   1:  PR[91,2] = PR[90,2] + -1.776;
   1:L PR[91] R[100]mm/sec CNT100TB   .50sec,CALL END_PUD;
   1:  PR[92] = PR[91];
   1:  PR[92,3] = PR[92,3] + 20;
   1:J PR[92] 10% FINE;
   1:  PR[91] = PR[90];
   1:  PR[91,1] = PR[90,1] + 4.469;
   1:  PR[91,2] = PR[90,2] + -0.729;
   1:  PR[91,3] = PR[90,3] + 32.695;
   1:  PR[92] = PR[91];
   1:  PR[92,3] = PR[92,3] + 20;
   1:J PR[92] 10% FINE;
   1:L PR[91] R[100]mm/sec CNT100;
   1:  CALL LASER_DRAHT_START;
   1:  PR[91,1] = PR[90,1] + 5.143;
   1:  PR[91,2] = PR[90,2] + -5.829;
   1:L PR[91] R[100]mm/sec CNT100;
   1:  PR[91,1] = PR[90,1] + 7.118;
   1:  PR[91,2] = PR[90,2] + -10.577;
   1:L PR[91] R[100]mm/sec CNT100;
   1:  PR[91,1] = PR[90,1] + 10.256;
   1:  PR[91,2] = PR[90,2] + -14.648;
   1:L PR[91] R[100]mm/sec CNT100;
   1:  PR[91,1] = PR[90,1] + 14.340;
   1:  PR[91,2] = PR[90,2] + -17.763;
   1:L PR[91] R[100]mm/sec CNT100;
   1:  PR[91,1] = PR[90,1] + 17.726;
   1:  PR[91,2] = PR[90,2] + -19.159;
   1:L PR[91] R[100]mm/sec CNT100;
   1:  PR[91,1] = PR[90,1] + 19.081;
   1:  PR[91,2] = PR[90,2] + -19.714;
   1:L PR[91] R[100]mm/sec CNT100;
   1:  PR[91,1] = PR[90,1] + 24.162;
   1:  PR[91,2] = PR[90,2] + -20.375;
   1:L PR[91] R[100]mm/sec CNT100;
   1:  PR[91,1] = PR[90,1] + 29.234;
   1:  PR[91,2] = PR[90,2] + -19.704;
   1:L PR[91] R[100]mm/sec CNT100;
   1:  PR[91,1] = PR[90,1] + 32.324;
   1:  PR[91,2] = PR[90,2] + -18.438;
   1:L PR[91] R[100]mm/sec CNT100;
   1:  PR[91,1] = PR[90,1] + 33.950;
   1:  PR[91,2] = PR[90,2] + -17.758;
   1:L PR[91] R[100]mm/sec CNT100;
   1:  PR[91,1] = PR[90,1] + 36.544;
   1:  PR[91,2] = PR[90,2] + -15.795;
   1:L PR[91] R[100]mm/sec CNT100;
   1:  PR[91,1] = PR[90,1] + 38.003;
   1:  PR[91,2] = PR[90,2] + -14.670;
   1:L PR[91] R[100]mm/sec CNT100;
   1:  PR[91,1] = PR[90,1] + 39.978;
   1:  PR[91,2] = PR[90,2] + -12.142;
   1:L PR[91] R[100]mm/sec CNT100;
   1:  PR[91,1] = PR[90,1] + 41.183;
   1:  PR[91,2] = PR[90,2] + -10.565;
   1:L PR[91] R[100]mm/sec CNT100;
   1:  PR[91,1] = PR[90,1] + 41.364;
   1:  PR[91,2] = PR[90,2] + -10.235;
   1:L PR[91] R[100]mm/sec CNT100;
   1:  PR[91,1] = PR[90,1] + 42.070;
   1:  PR[91,2] = PR[90,2] + -8.524;
   1:L PR[91] R[100]mm/sec CNT100;
   1:  PR[91,1] = PR[90,1] + 42.766;
   1:  PR[91,2] = PR[90,2] + -6.971;
   1:L PR[91] R[100]mm/sec CNT100;
   1:  PR[91,1] = PR[90,1] + 43.473;
   1:  PR[91,2] = PR[90,2] + -4.203;
   1:L PR[91] R[100]mm/sec CNT100;
   1:  PR[91,1] = PR[90,1] + 43.657;
   1:  PR[91,2] = PR[90,2] + -2.266;
   1:L PR[91] R[100]mm/sec CNT100;
   1:  PR[91,1] = PR[90,1] + 47.140;
   1:  PR[91,2] = PR[90,2] + -2.119;
   1:L PR[91] R[100]mm/sec CNT100;
   1:  PR[91,1] = PR[90,1] + 47.551;
   1:  PR[91,2] = PR[90,2] + -4.387;
   1:L PR[91] R[100]mm/sec CNT100;
   1:  PR[91,1] = PR[90,1] + 47.975;
   1:  PR[91,2] = PR[90,2] + -5.947;
   1:L PR[91] R[100]mm/sec CNT100;
   1:  PR[91,1] = PR[90,1] + 48.962;
   1:  PR[91,2] = PR[90,2] + -7.849;
   1:L PR[91] R[100]mm/sec CNT100;
   1:  PR[91,1] = PR[90,1] + 50.226;
   1:  PR[91,2] = PR[90,2] + -10.536;
   1:L PR[91] R[100]mm/sec CNT100;
   1:  PR[91,1] = PR[90,1] + 50.408;
   1:  PR[91,2] = PR[90,2] + -10.773;
   1:L PR[91] R[100]mm/sec CNT100;
   1:  PR[91,1] = PR[90,1] + 53.451;
   1:  PR[91,2] = PR[90,2] + -14.307;
   1:L PR[91] R[100]mm/sec CNT100;
   1:  PR[91,1] = PR[90,1] + 54.867;
   1:  PR[91,2] = PR[90,2] + -15.442;
   1:L PR[91] R[100]mm/sec CNT100;
   1:  PR[91,1] = PR[90,1] + 57.318;
   1:  PR[91,2] = PR[90,2] + -17.146;
   1:L PR[91] R[100]mm/sec CNT100;
   1:  PR[91,1] = PR[90,1] + 60.422;
   1:  PR[91,2] = PR[90,2] + -18.651;
   1:L PR[91] R[100]mm/sec CNT100;
   1:  PR[91,1] = PR[90,1] + 61.529;
   1:  PR[91,2] = PR[90,2] + -19.083;
   1:L PR[91] R[100]mm/sec CNT100;
   1:  PR[91,1] = PR[90,1] + 65.504;
   1:  PR[91,2] = PR[90,2] + -20.053;
   1:L PR[91] R[100]mm/sec CNT100;
   1:  PR[91,1] = PR[90,1] + 66.069;
   1:  PR[91,2] = PR[90,2] + -20.209;
   1:L PR[91] R[100]mm/sec CNT100;
   1:  PR[91,1] = PR[90,1] + 70.771;
   1:  PR[91,2] = PR[90,2] + -20.477;
   1:L PR[91] R[100]mm/sec CNT100;
   1:  PR[91,1] = PR[90,1] + 71.856;
   1:  PR[91,2] = PR[90,2] + -20.322;
   1:L PR[91] R[100]mm/sec CNT100;
   1:  PR[91,1] = PR[90,1] + 75.350;
   1:  PR[91,2] = PR[90,2] + -19.774;
   1:L PR[91] R[100]mm/sec CNT100;
   1:  PR[91,1] = PR[90,1] + 77.247;
   1:  PR[91,2] = PR[90,2] + -19.075;
   1:L PR[91] R[100]mm/sec CNT100;
   1:  PR[91,1] = PR[90,1] + 79.618;
   1:  PR[91,2] = PR[90,2] + -18.166;
   1:L PR[91] R[100]mm/sec CNT100;
   1:  PR[91,1] = PR[90,1] + 81.915;
   1:  PR[91,2] = PR[90,2] + -16.702;
   1:L PR[91] R[100]mm/sec CNT100;
   1:  PR[91,1] = PR[90,1] + 83.382;
   1:  PR[91,2] = PR[90,2] + -15.743;
   1:L PR[91] R[100]mm/sec CNT100;
   1:  PR[91,1] = PR[90,1] + 86.493;
   1:  PR[91,2] = PR[90,2] + -12.622;
   1:L PR[91] R[100]mm/sec CNT100;
   1:  PR[91,1] = PR[90,1] + 88.806;
   1:  PR[91,2] = PR[90,2] + -8.967;
   1:L PR[91] R[100]mm/sec CNT100;
   1:  PR[91,1] = PR[90,1] + 90.231;
   1:  PR[91,2] = PR[90,2] + -4.940;
   1:L PR[91] R[100]mm/sec CNT100;
   1:  PR[91,1] = PR[90,1] + 90.718;
   1:  PR[91,2] = PR[90,2] + -0.729;
   1:L PR[91] R[100]mm/sec CNT100;
   1:  PR[91,1] = PR[90,1] + 90.231;
   1:  PR[91,2] = PR[90,2] + 3.481;
   1:L PR[91] R[100]mm/sec CNT100;
   1:  PR[91,1] = PR[90,1] + 88.806;
   1:  PR[91,2] = PR[90,2] + 7.508;
   1:L PR[91] R[100]mm/sec CNT100;
   1:  PR[91,1] = PR[90,1] + 86.495;
   1:  PR[91,2] = PR[90,2] + 11.160;
   1:L PR[91] R[100]mm/sec CNT100;
   1:  PR[91,1] = PR[90,1] + 84.284;
   1:  PR[91,2] = PR[90,2] + 13.362;
   1:L PR[91] R[100]mm/sec CNT100;
   1:  PR[91,1] = PR[90,1] + 83.384;
   1:  PR[91,2] = PR[90,2] + 14.279;
   1:L PR[91] R[100]mm/sec CNT100;
   1:  PR[91,1] = PR[90,1] + 81.098;
   1:  PR[91,2] = PR[90,2] + 15.732;
   1:L PR[91] R[100]mm/sec CNT100;
   1:  PR[91,1] = PR[90,1] + 79.618;
   1:  PR[91,2] = PR[90,2] + 16.704;
   1:L PR[91] R[100]mm/sec CNT100;
   1:  PR[91,1] = PR[90,1] + 77.562;
   1:  PR[91,2] = PR[90,2] + 17.457;
   1:L PR[91] R[100]mm/sec CNT100;
   1:  PR[91,1] = PR[90,1] + 75.350;
   1:  PR[91,2] = PR[90,2] + 18.312;
   1:L PR[91] R[100]mm/sec CNT100;
   1:  PR[91,1] = PR[90,1] + 73.814;
   1:  PR[91,2] = PR[90,2] + 18.527;
   1:L PR[91] R[100]mm/sec CNT100;
   1:  PR[91,1] = PR[90,1] + 70.770;
   1:  PR[91,2] = PR[90,2] + 19.014;
   1:L PR[91] R[100]mm/sec CNT100;
   1:  PR[91,1] = PR[90,1] + 69.982;
   1:  PR[91,2] = PR[90,2] + 18.956;
   1:L PR[91] R[100]mm/sec CNT100;
   1:  PR[91,1] = PR[90,1] + 66.065;
   1:  PR[91,2] = PR[90,2] + 18.749;
   1:L PR[91] R[100]mm/sec CNT100;
   1:  PR[91,1] = PR[90,1] + 65.504;
   1:  PR[91,2] = PR[90,2] + 18.594;
   1:L PR[91] R[100]mm/sec CNT100;
   1:  PR[91,1] = PR[90,1] + 61.529;
   1:  PR[91,2] = PR[90,2] + 17.625;
   1:L PR[91] R[100]mm/sec CNT100;
   1:  PR[91,1] = PR[90,1] + 60.422;
   1:  PR[91,2] = PR[90,2] + 17.192;
   1:L PR[91] R[100]mm/sec CNT100;
   1:  PR[91,1] = PR[90,1] + 57.318;
   1:  PR[91,2] = PR[90,2] + 15.687;
   1:L PR[91] R[100]mm/sec CNT100;
   1:  PR[91,1] = PR[90,1] + 54.868;
   1:  PR[91,2] = PR[90,2] + 13.984;
   1:L PR[91] R[100]mm/sec CNT100;
   1:  PR[91,1] = PR[90,1] + 53.452;
   1:  PR[91,2] = PR[90,2] + 12.849;
   1:L PR[91] R[100]mm/sec CNT100;
   1:  PR[91,1] = PR[90,1] + 50.409;
   1:  PR[91,2] = PR[90,2] + 9.316;
   1:L PR[91] R[100]mm/sec CNT100;
   1:  PR[91,1] = PR[90,1] + 50.226;
   1:  PR[91,2] = PR[90,2] + 9.078;
   1:L PR[91] R[100]mm/sec CNT100;
   1:  PR[91,1] = PR[90,1] + 48.961;
   1:  PR[91,2] = PR[90,2] + 6.389;
   1:L PR[91] R[100]mm/sec CNT100;
   1:  PR[91,1] = PR[90,1] + 47.985;
   1:  PR[91,2] = PR[90,2] + 4.511;
   1:L PR[91] R[100]mm/sec CNT100;
   1:  PR[91,1] = PR[90,1] + 47.482;
   1:  PR[91,2] = PR[90,2] + 2.646;
   1:L PR[91] R[100]mm/sec CNT100;
   1:  PR[91,1] = PR[90,1] + 47.137;
   1:  PR[91,2] = PR[90,2] + 0.760;
   1:L PR[91] R[100]mm/sec CNT100;
   1:  PR[91,1] = PR[90,1] + 43.653;
   1:  PR[91,2] = PR[90,2] + 0.914;
   1:L PR[91] R[100]mm/sec CNT100;
   1:  PR[91,1] = PR[90,1] + 43.495;
   1:  PR[91,2] = PR[90,2] + 2.623;
   1:L PR[91] R[100]mm/sec CNT100;
   1:  PR[91,1] = PR[90,1] + 42.693;
   1:  PR[91,2] = PR[90,2] + 5.724;
   1:L PR[91] R[100]mm/sec CNT100;
   1:  PR[91,1] = PR[90,1] + 42.326;
   1:  PR[91,2] = PR[90,2] + 6.613;
   1:L PR[91] R[100]mm/sec CNT100;
   1:  PR[91,1] = PR[90,1] + 41.404;
   1:  PR[91,2] = PR[90,2] + 8.700;
   1:L PR[91] R[100]mm/sec CNT100;
   1:  PR[91,1] = PR[90,1] + 41.184;
   1:  PR[91,2] = PR[90,2] + 9.104;
   1:L PR[91] R[100]mm/sec CNT100;
   1:  PR[91,1] = PR[90,1] + 39.948;
   1:  PR[91,2] = PR[90,2] + 10.732;
   1:L PR[91] R[100]mm/sec CNT100;
   1:  PR[91,1] = PR[90,1] + 37.982;
   1:  PR[91,2] = PR[90,2] + 13.232;
   1:L PR[91] R[100]mm/sec CNT100;
   1:  PR[91,1] = PR[90,1] + 36.524;
   1:  PR[91,2] = PR[90,2] + 14.357;
   1:L PR[91] R[100]mm/sec CNT100;
   1:  PR[91,1] = PR[90,1] + 33.926;
   1:  PR[91,2] = PR[90,2] + 16.313;
   1:L PR[91] R[100]mm/sec CNT100;
   1:  PR[91,1] = PR[90,1] + 32.300;
   1:  PR[91,2] = PR[90,2] + 16.993;
   1:L PR[91] R[100]mm/sec CNT100;
   1:  PR[91,1] = PR[90,1] + 29.208;
   1:  PR[91,2] = PR[90,2] + 18.253;
   1:L PR[91] R[100]mm/sec CNT100;
   1:  PR[91,1] = PR[90,1] + 27.552;
   1:  PR[91,2] = PR[90,2] + 18.478;
   1:L PR[91] R[100]mm/sec CNT100;
   1:  PR[91,1] = PR[90,1] + 24.143;
   1:  PR[91,2] = PR[90,2] + 18.917;
   1:L PR[91] R[100]mm/sec CNT100;
   1:  PR[91,1] = PR[90,1] + 19.065;
   1:  PR[91,2] = PR[90,2] + 18.251;
   1:L PR[91] R[100]mm/sec CNT100;
   1:  PR[91,1] = PR[90,1] + 14.324;
   1:  PR[91,2] = PR[90,2] + 16.295;
   1:L PR[91] R[100]mm/sec CNT100;
   1:  PR[91,1] = PR[90,1] + 13.237;
   1:  PR[91,2] = PR[90,2] + 15.467;
   1:L PR[91] R[100]mm/sec CNT100;
   1:  PR[91,1] = PR[90,1] + 10.248;
   1:  PR[91,2] = PR[90,2] + 13.181;
   1:L PR[91] R[100]mm/sec CNT100;
   1:  PR[91,1] = PR[90,1] + 7.114;
   1:  PR[91,2] = PR[90,2] + 9.111;
   1:L PR[91] R[100]mm/sec CNT100;
   1:  PR[91,1] = PR[90,1] + 5.142;
   1:  PR[91,2] = PR[90,2] + 4.367;
   1:L PR[91] R[100]mm/sec CNT100;
   1:  PR[91,1] = PR[90,1] + 4.469;
   1:  PR[91,2] = PR[90,2] + -0.729;
   1:L PR[91] R[100]mm/sec CNT100TB   .50sec,CALL END_PUD;
   1:  PR[92] = PR[91];
   1:  PR[92,3] = PR[92,3] + 20;
   1:J PR[92] 10% FINE;
   1:  PR[91,1] = PR[90,1] + -41.681;
   1:  PR[91,2] = PR[90,2] + -0.717;
   1:  PR[92] = PR[91];
   1:  PR[92,3] = PR[92,3] + 20;
   1:J PR[92] 10% FINE;
   1:L PR[91] R[100]mm/sec CNT100;
   1:  CALL LASER_DRAHT_START;
   1:  PR[91,1] = PR[90,1] + -41.546;
   1:  PR[91,2] = PR[90,2] + -1.807;
   1:L PR[91] R[100]mm/sec CNT100;
   1:  PR[91,1] = PR[90,1] + -41.199;
   1:  PR[91,2] = PR[90,2] + -4.905;
   1:L PR[91] R[100]mm/sec CNT100;
   1:  PR[91,1] = PR[90,1] + -39.815;
   1:  PR[91,2] = PR[90,2] + -8.880;
   1:L PR[91] R[100]mm/sec CNT100;
   1:  PR[91,1] = PR[90,1] + -37.577;
   1:  PR[91,2] = PR[90,2] + -12.464;
   1:L PR[91] R[100]mm/sec CNT100;
   1:  PR[91,1] = PR[90,1] + -34.591;
   1:  PR[91,2] = PR[90,2] + -15.481;
   1:L PR[91] R[100]mm/sec CNT100;
   1:  PR[91,1] = PR[90,1] + -30.997;
   1:  PR[91,2] = PR[90,2] + -17.783;
   1:L PR[91] R[100]mm/sec CNT100;
   1:  PR[91,1] = PR[90,1] + -26.963;
   1:  PR[91,2] = PR[90,2] + -19.248;
   1:L PR[91] R[100]mm/sec CNT100;
   1:  PR[91,1] = PR[90,1] + -22.671;
   1:  PR[91,2] = PR[90,2] + -19.803;
   1:L PR[91] R[100]mm/sec CNT100;
   1:  PR[91,1] = PR[90,1] + -18.279;
   1:  PR[91,2] = PR[90,2] + -19.439;
   1:L PR[91] R[100]mm/sec CNT100;
   1:  PR[91,1] = PR[90,1] + -18.066;
   1:  PR[91,2] = PR[90,2] + -19.387;
   1:L PR[91] R[100]mm/sec CNT100;
   1:  PR[91,1] = PR[90,1] + -14.122;
   1:  PR[91,2] = PR[90,2] + -18.164;
   1:L PR[91] R[100]mm/sec CNT100;
   1:  PR[91,1] = PR[90,1] + -13.522;
   1:  PR[91,2] = PR[90,2] + -17.867;
   1:L PR[91] R[100]mm/sec CNT100;
   1:  PR[91,1] = PR[90,1] + -10.339;
   1:  PR[91,2] = PR[90,2] + -16.033;
   1:L PR[91] R[100]mm/sec CNT100;
   1:  PR[91,1] = PR[90,1] + -9.487;
   1:  PR[91,2] = PR[90,2] + -15.341;
   1:L PR[91] R[100]mm/sec CNT100;
   1:  PR[91,1] = PR[90,1] + -7.115;
   1:  PR[91,2] = PR[90,2] + -13.139;
   1:L PR[91] R[100]mm/sec CNT100;
   1:  PR[91,1] = PR[90,1] + -6.219;
   1:  PR[91,2] = PR[90,2] + -11.981;
   1:L PR[91] R[100]mm/sec CNT100;
   1:  PR[91,1] = PR[90,1] + -4.619;
   1:  PR[91,2] = PR[90,2] + -9.603;
   1:L PR[91] R[100]mm/sec CNT100;
   1:  PR[91,1] = PR[90,1] + -3.902;
   1:  PR[91,2] = PR[90,2] + -8.021;
   1:L PR[91] R[100]mm/sec CNT100;
   1:  PR[91,1] = PR[90,1] + -2.996;
   1:  PR[91,2] = PR[90,2] + -5.591;
   1:L PR[91] R[100]mm/sec CNT100;
   1:  PR[91,1] = PR[90,1] + -2.643;
   1:  PR[91,2] = PR[90,2] + -3.715;
   1:L PR[91] R[100]mm/sec CNT100;
   1:  PR[91,1] = PR[90,1] + -2.344;
   1:  PR[91,2] = PR[90,2] + -1.237;
   1:L PR[91] R[100]mm/sec CNT100;
   1:  PR[91,1] = PR[90,1] + -2.332;
   1:  PR[91,2] = PR[90,2] + -0.821;
   1:L PR[91] R[100]mm/sec CNT100;
   1:  PR[91,1] = PR[90,1] + -2.639;
   1:  PR[91,2] = PR[90,2] + 1.729;
   1:L PR[91] R[100]mm/sec CNT100;
   1:  PR[91,1] = PR[90,1] + -2.659;
   1:  PR[91,2] = PR[90,2] + 2.337;
   1:L PR[91] R[100]mm/sec CNT100;
   1:  PR[91,1] = PR[90,1] + -2.994;
   1:  PR[91,2] = PR[90,2] + 4.125;
   1:L PR[91] R[100]mm/sec CNT100;
   1:  PR[91,1] = PR[90,1] + -3.900;
   1:  PR[91,2] = PR[90,2] + 6.556;
   1:L PR[91] R[100]mm/sec CNT100;
   1:  PR[91,1] = PR[90,1] + -4.616;
   1:  PR[91,2] = PR[90,2] + 8.139;
   1:L PR[91] R[100]mm/sec CNT100;
   1:  PR[91,1] = PR[90,1] + -6.216;
   1:  PR[91,2] = PR[90,2] + 10.518;
   1:L PR[91] R[100]mm/sec CNT100;
   1:  PR[91,1] = PR[90,1] + -7.112;
   1:  PR[91,2] = PR[90,2] + 11.677;
   1:L PR[91] R[100]mm/sec CNT100;
   1:  PR[91,1] = PR[90,1] + -9.484;
   1:  PR[91,2] = PR[90,2] + 13.879;
   1:L PR[91] R[100]mm/sec CNT100;
   1:  PR[91,1] = PR[90,1] + -10.336;
   1:  PR[91,2] = PR[90,2] + 14.573;
   1:L PR[91] R[100]mm/sec CNT100;
   1:  PR[91,1] = PR[90,1] + -13.520;
   1:  PR[91,2] = PR[90,2] + 16.407;
   1:L PR[91] R[100]mm/sec CNT100;
   1:  PR[91,1] = PR[90,1] + -14.120;
   1:  PR[91,2] = PR[90,2] + 16.705;
   1:L PR[91] R[100]mm/sec CNT100;
   1:  PR[91,1] = PR[90,1] + -18.065;
   1:  PR[91,2] = PR[90,2] + 17.927;
   1:L PR[91] R[100]mm/sec CNT100;
   1:  PR[91,1] = PR[90,1] + -18.278;
   1:  PR[91,2] = PR[90,2] + 17.980;
   1:L PR[91] R[100]mm/sec CNT100;
   1:  PR[91,1] = PR[90,1] + -22.679;
   1:  PR[91,2] = PR[90,2] + 18.344;
   1:L PR[91] R[100]mm/sec CNT100;
   1:  PR[91,1] = PR[90,1] + -26.963;
   1:  PR[91,2] = PR[90,2] + 17.790;
   1:L PR[91] R[100]mm/sec CNT100;
   1:  PR[91,1] = PR[90,1] + -30.997;
   1:  PR[91,2] = PR[90,2] + 16.324;
   1:L PR[91] R[100]mm/sec CNT100;
   1:  PR[91,1] = PR[90,1] + -34.591;
   1:  PR[91,2] = PR[90,2] + 14.022;
   1:L PR[91] R[100]mm/sec CNT100;
   1:  PR[91,1] = PR[90,1] + -37.577;
   1:  PR[91,2] = PR[90,2] + 11.005;
   1:L PR[91] R[100]mm/sec CNT100;
   1:  PR[91,1] = PR[90,1] + -39.815;
   1:  PR[91,2] = PR[90,2] + 7.422;
   1:L PR[91] R[100]mm/sec CNT100;
   1:  PR[91,1] = PR[90,1] + -41.199;
   1:  PR[91,2] = PR[90,2] + 3.445;
   1:L PR[91] R[100]mm/sec CNT100;
   1:  PR[91,1] = PR[90,1] + -41.330;
   1:  PR[91,2] = PR[90,2] + 2.291;
   1:L PR[91] R[100]mm/sec CNT100;
   1:  PR[91,1] = PR[90,1] + -41.361;
   1:  PR[91,2] = PR[90,2] + 2.140;
   1:L PR[91] R[100]mm/sec CNT100;
   1:  PR[91,1] = PR[90,1] + -41.681;
   1:  PR[91,2] = PR[90,2] + -0.717;
   1:L PR[91] R[100]mm/sec CNT100TB   .50sec,CALL END_PUD;
   1:  PR[92] = PR[91];
   1:  PR[92,3] = PR[92,3] + 20;
   1:J PR[92] 10% FINE;
   1:  PR[91,1] = PR[90,1] + -77.314;
   1:  PR[91,2] = PR[90,2] + -18.642;
   1:  PR[92] = PR[91];
   1:  PR[92,3] = PR[92,3] + 20;
   1:J PR[92] 10% FINE;
   1:L PR[91] R[100]mm/sec CNT100;
   1:  CALL LASER_DRAHT_START;
   1:  PR[91,1] = PR[90,1] + -74.683;
   1:  PR[91,2] = PR[90,2] + -19.231;
   1:L PR[91] R[100]mm/sec CNT100;
   1:  PR[91,1] = PR[90,1] + -73.251;
   1:  PR[91,2] = PR[90,2] + -19.573;
   1:L PR[91] R[100]mm/sec CNT100;
   1:  PR[91,1] = PR[90,1] + -71.069;
   1:  PR[91,2] = PR[90,2] + -19.621;
   1:L PR[91] R[100]mm/sec CNT100;
   1:  PR[91,1] = PR[90,1] + -69.047;
   1:  PR[91,2] = PR[90,2] + -19.694;
   1:L PR[91] R[100]mm/sec CNT100;
   1:  PR[91,1] = PR[90,1] + -67.474;
   1:  PR[91,2] = PR[90,2] + -19.413;
   1:L PR[91] R[100]mm/sec CNT100;
   1:  PR[91,1] = PR[90,1] + -64.878;
   1:  PR[91,2] = PR[90,2] + -18.989;
   1:L PR[91] R[100]mm/sec CNT100;
   1:  PR[91,1] = PR[90,1] + -63.990;
   1:  PR[91,2] = PR[90,2] + -18.636;
   1:L PR[91] R[100]mm/sec CNT100;
   1:  PR[91,1] = PR[90,1] + -60.914;
   1:  PR[91,2] = PR[90,2] + -17.467;
   1:L PR[91] R[100]mm/sec CNT100;
   1:  PR[91,1] = PR[90,1] + -58.205;
   1:  PR[91,2] = PR[90,2] + -15.726;
   1:L PR[91] R[100]mm/sec CNT100;
   1:  PR[91,1] = PR[90,1] + -57.250;
   1:  PR[91,2] = PR[90,2] + -15.156;
   1:L PR[91] R[100]mm/sec CNT100;
   1:  PR[91,1] = PR[90,1] + -54.565;
   1:  PR[91,2] = PR[90,2] + -12.649;
   1:L PR[91] R[100]mm/sec CNT100;
   1:  PR[91,1] = PR[90,1] + -54.071;
   1:  PR[91,2] = PR[90,2] + -12.203;
   1:L PR[91] R[100]mm/sec CNT100;
   1:  PR[91,1] = PR[90,1] + -52.386;
   1:  PR[91,2] = PR[90,2] + -9.733;
   1:L PR[91] R[100]mm/sec CNT100;
   1:  PR[91,1] = PR[90,1] + -51.665;
   1:  PR[91,2] = PR[90,2] + -8.704;
   1:L PR[91] R[100]mm/sec CNT100;
   1:  PR[91,1] = PR[90,1] + -50.168;
   1:  PR[91,2] = PR[90,2] + -4.823;
   1:L PR[91] R[100]mm/sec CNT100;
   1:  PR[91,1] = PR[90,1] + -49.910;
   1:  PR[91,2] = PR[90,2] + -2.744;
   1:L PR[91] R[100]mm/sec CNT100;
   1:  PR[91,1] = PR[90,1] + -49.770;
   1:  PR[91,2] = PR[90,2] + -0.743;
   1:L PR[91] R[100]mm/sec CNT100;
   1:  PR[91,1] = PR[90,1] + -49.798;
   1:  PR[91,2] = PR[90,2] + -0.406;
   1:L PR[91] R[100]mm/sec CNT100;
   1:  PR[91,1] = PR[90,1] + -50.252;
   1:  PR[91,2] = PR[90,2] + 3.373;
   1:L PR[91] R[100]mm/sec CNT100;
   1:  PR[91,1] = PR[90,1] + -51.720;
   1:  PR[91,2] = PR[90,2] + 7.273;
   1:L PR[91] R[100]mm/sec CNT100;
   1:  PR[91,1] = PR[90,1] + -52.373;
   1:  PR[91,2] = PR[90,2] + 8.257;
   1:L PR[91] R[100]mm/sec CNT100;
   1:  PR[91,1] = PR[90,1] + -54.073;
   1:  PR[91,2] = PR[90,2] + 10.775;
   1:L PR[91] R[100]mm/sec CNT100;
   1:  PR[91,1] = PR[90,1] + -55.593;
   1:  PR[91,2] = PR[90,2] + 12.234;
   1:L PR[91] R[100]mm/sec CNT100;
   1:  PR[91,1] = PR[90,1] + -57.173;
   1:  PR[91,2] = PR[90,2] + 13.722;
   1:L PR[91] R[100]mm/sec CNT100;
   1:  PR[91,1] = PR[90,1] + -60.872;
   1:  PR[91,2] = PR[90,2] + 15.996;
   1:L PR[91] R[100]mm/sec CNT100;
   1:  PR[91,1] = PR[90,1] + -64.984;
   1:  PR[91,2] = PR[90,2] + 17.505;
   1:L PR[91] R[100]mm/sec CNT100;
   1:  PR[91,1] = PR[90,1] + -69.137;
   1:  PR[91,2] = PR[90,2] + 18.221;
   1:L PR[91] R[100]mm/sec CNT100;
   1:  PR[91,1] = PR[90,1] + -73.297;
   1:  PR[91,2] = PR[90,2] + 18.107;
   1:L PR[91] R[100]mm/sec CNT100;
   1:  PR[91,1] = PR[90,1] + -77.320;
   1:  PR[91,2] = PR[90,2] + 17.184;
   1:L PR[91] R[100]mm/sec CNT100;
   1:  PR[91,1] = PR[90,1] + -81.037;
   1:  PR[91,2] = PR[90,2] + 15.500;
   1:L PR[91] R[100]mm/sec CNT100;
   1:  PR[91,1] = PR[90,1] + -84.300;
   1:  PR[91,2] = PR[90,2] + 13.138;
   1:L PR[91] R[100]mm/sec CNT100;
   1:  PR[91,1] = PR[90,1] + -86.977;
   1:  PR[91,2] = PR[90,2] + 10.199;
   1:L PR[91] R[100]mm/sec CNT100;
   1:  PR[91,1] = PR[90,1] + -88.967;
   1:  PR[91,2] = PR[90,2] + 6.813;
   1:L PR[91] R[100]mm/sec CNT100;
   1:  PR[91,1] = PR[90,1] + -90.190;
   1:  PR[91,2] = PR[90,2] + 3.119;
   1:L PR[91] R[100]mm/sec CNT100;
   1:  PR[91,1] = PR[90,1] + -90.556;
   1:  PR[91,2] = PR[90,2] + -0.259;
   1:L PR[91] R[100]mm/sec CNT100;
   1:  PR[91,1] = PR[90,1] + -90.654;
   1:  PR[91,2] = PR[90,2] + -0.746;
   1:L PR[91] R[100]mm/sec CNT100;
   1:  PR[91,1] = PR[90,1] + -90.252;
   1:  PR[91,2] = PR[90,2] + -4.584;
   1:L PR[91] R[100]mm/sec CNT100;
   1:  PR[91,1] = PR[90,1] + -89.055;
   1:  PR[91,2] = PR[90,2] + -8.268;
   1:L PR[91] R[100]mm/sec CNT100;
   1:  PR[91,1] = PR[90,1] + -87.060;
   1:  PR[91,2] = PR[90,2] + -11.645;
   1:L PR[91] R[100]mm/sec CNT100;
   1:  PR[91,1] = PR[90,1] + -84.363;
   1:  PR[91,2] = PR[90,2] + -14.584;
   1:L PR[91] R[100]mm/sec CNT100;
   1:  PR[91,1] = PR[90,1] + -81.074;
   1:  PR[91,2] = PR[90,2] + -16.950;
   1:L PR[91] R[100]mm/sec CNT100;
   1:  PR[91,1] = PR[90,1] + -78.209;
   1:  PR[91,2] = PR[90,2] + -18.229;
   1:L PR[91] R[100]mm/sec CNT100;
   1:  PR[91,1] = PR[90,1] + -77.314;
   1:  PR[91,2] = PR[90,2] + -18.642;
   1:L PR[91] R[100]mm/sec CNT100TB   .50sec,CALL END_PUD;
   1:  PR[92] = PR[91];
   1:  PR[92,3] = PR[92,3] + 20;
   1:J PR[92] 10% FINE;
   1:  PR[91] = PR[90];
   1:  PR[91,1] = PR[90,1] + 4.937;
   1:  PR[91,2] = PR[90,2] + -5.866;
   1:  PR[91,3] = PR[90,3] + 33.995;
   1:  PR[92] = PR[91];
   1:  PR[92,3] = PR[92,3] + 20;
   1:J PR[92] 10% FINE;
   1:L PR[91] R[100]mm/sec CNT100;
   1:  CALL LASER_DRAHT_START;
   1:  PR[91,1] = PR[90,1] + 6.927;
   1:  PR[91,2] = PR[90,2] + -10.647;
   1:L PR[91] R[100]mm/sec CNT100;
   1:  PR[91,1] = PR[90,1] + 10.086;
   1:  PR[91,2] = PR[90,2] + -14.747;
   1:L PR[91] R[100]mm/sec CNT100;
   1:  PR[91,1] = PR[90,1] + 14.198;
   1:  PR[91,2] = PR[90,2] + -17.884;
   1:L PR[91] R[100]mm/sec CNT100;
   1:  PR[91,1] = PR[90,1] + 18.974;
   1:  PR[91,2] = PR[90,2] + -19.851;
   1:L PR[91] R[100]mm/sec CNT100;
   1:  PR[91,1] = PR[90,1] + 24.089;
   1:  PR[91,2] = PR[90,2] + -20.518;
   1:L PR[91] R[100]mm/sec CNT100;
   1:  PR[91,1] = PR[90,1] + 28.004;
   1:  PR[91,2] = PR[90,2] + -20.007;
   1:L PR[91] R[100]mm/sec CNT100;
   1:  PR[91,1] = PR[90,1] + 29.188;
   1:  PR[91,2] = PR[90,2] + -19.846;
   1:L PR[91] R[100]mm/sec CNT100;
   1:  PR[91,1] = PR[90,1] + 33.946;
   1:  PR[91,2] = PR[90,2] + -17.886;
   1:L PR[91] R[100]mm/sec CNT100;
   1:  PR[91,1] = PR[90,1] + 36.932;
   1:  PR[91,2] = PR[90,2] + -15.626;
   1:L PR[91] R[100]mm/sec CNT100;
   1:  PR[91,1] = PR[90,1] + 38.023;
   1:  PR[91,2] = PR[90,2] + -14.784;
   1:L PR[91] R[100]mm/sec CNT100;
   1:  PR[91,1] = PR[90,1] + 40.305;
   1:  PR[91,2] = PR[90,2] + -11.865;
   1:L PR[91] R[100]mm/sec CNT100;
   1:  PR[91,1] = PR[90,1] + 41.228;
   1:  PR[91,2] = PR[90,2] + -10.656;
   1:L PR[91] R[100]mm/sec CNT100;
   1:  PR[91,1] = PR[90,1] + 41.454;
   1:  PR[91,2] = PR[90,2] + -10.245;
   1:L PR[91] R[100]mm/sec CNT100;
   1:  PR[91,1] = PR[90,1] + 41.969;
   1:  PR[91,2] = PR[90,2] + -8.998;
   1:L PR[91] R[100]mm/sec CNT100;
   1:  PR[91,1] = PR[90,1] + 42.774;
   1:  PR[91,2] = PR[90,2] + -7.199;
   1:L PR[91] R[100]mm/sec CNT100;
   1:  PR[91,1] = PR[90,1] + 44.425;
   1:  PR[91,2] = PR[90,2] + -0.731;
   1:L PR[91] R[100]mm/sec CNT100;
   1:  PR[91,1] = PR[90,1] + 42.691;
   1:  PR[91,2] = PR[90,2] + 5.979;
   1:L PR[91] R[100]mm/sec CNT100;
   1:  PR[91,1] = PR[90,1] + 42.559;
   1:  PR[91,2] = PR[90,2] + 6.299;
   1:L PR[91] R[100]mm/sec CNT100;
   1:  PR[91,1] = PR[90,1] + 41.498;
   1:  PR[91,2] = PR[90,2] + 8.701;
   1:L PR[91] R[100]mm/sec CNT100;
   1:  PR[91,1] = PR[90,1] + 41.229;
   1:  PR[91,2] = PR[90,2] + 9.195;
   1:L PR[91] R[100]mm/sec CNT100;
   1:  PR[91,1] = PR[90,1] + 40.269;
   1:  PR[91,2] = PR[90,2] + 10.462;
   1:L PR[91] R[100]mm/sec CNT100;
   1:  PR[91,1] = PR[90,1] + 37.999;
   1:  PR[91,2] = PR[90,2] + 13.349;
   1:L PR[91] R[100]mm/sec CNT100;
   1:  PR[91,1] = PR[90,1] + 36.907;
   1:  PR[91,2] = PR[90,2] + 14.192;
   1:L PR[91] R[100]mm/sec CNT100;
   1:  PR[91,1] = PR[90,1] + 33.914;
   1:  PR[91,2] = PR[90,2] + 16.446;
   1:L PR[91] R[100]mm/sec CNT100;
   1:  PR[91,1] = PR[90,1] + 32.719;
   1:  PR[91,2] = PR[90,2] + 16.946;
   1:L PR[91] R[100]mm/sec CNT100;
   1:  PR[91,1] = PR[90,1] + 29.163;
   1:  PR[91,2] = PR[90,2] + 18.395;
   1:L PR[91] R[100]mm/sec CNT100;
   1:  PR[91,1] = PR[90,1] + 27.976;
   1:  PR[91,2] = PR[90,2] + 18.556;
   1:L PR[91] R[100]mm/sec CNT100;
   1:  PR[91,1] = PR[90,1] + 24.065;
   1:  PR[91,2] = PR[90,2] + 19.059;
   1:L PR[91] R[100]mm/sec CNT100;
   1:  PR[91,1] = PR[90,1] + 18.954;
   1:  PR[91,2] = PR[90,2] + 18.386;
   1:L PR[91] R[100]mm/sec CNT100;
   1:  PR[91,1] = PR[90,1] + 14.183;
   1:  PR[91,2] = PR[90,2] + 16.417;
   1:L PR[91] R[100]mm/sec CNT100;
   1:  PR[91,1] = PR[90,1] + 10.077;
   1:  PR[91,2] = PR[90,2] + 13.279;
   1:L PR[91] R[100]mm/sec CNT100;
   1:  PR[91,1] = PR[90,1] + 6.922;
   1:  PR[91,2] = PR[90,2] + 9.181;
   1:L PR[91] R[100]mm/sec CNT100;
   1:  PR[91,1] = PR[90,1] + 4.936;
   1:  PR[91,2] = PR[90,2] + 4.403;
   1:L PR[91] R[100]mm/sec CNT100;
   1:  PR[91,1] = PR[90,1] + 4.259;
   1:  PR[91,2] = PR[90,2] + -0.729;
   1:L PR[91] R[100]mm/sec CNT100;
   1:  PR[91,1] = PR[90,1] + 4.937;
   1:  PR[91,2] = PR[90,2] + -5.866;
   1:L PR[91] R[100]mm/sec CNT100TB   .50sec,CALL END_PUD;
   1:  PR[92] = PR[91];
   1:  PR[92,3] = PR[92,3] + 20;
   1:J PR[92] 10% FINE;
   1:  PR[91,1] = PR[90,1] + 45.494;
   1:  PR[91,2] = PR[90,2] + -0.780;
   1:  PR[92] = PR[91];
   1:  PR[92,3] = PR[92,3] + 20;
   1:J PR[92] 10% FINE;
   1:L PR[91] R[100]mm/sec CNT100;
   1:  CALL LASER_DRAHT_START;
   1:  PR[91,1] = PR[90,1] + 47.117;
   1:  PR[91,2] = PR[90,2] + -6.749;
   1:L PR[91] R[100]mm/sec CNT100;
   1:  PR[91,1] = PR[90,1] + 49.050;
   1:  PR[91,2] = PR[90,2] + -10.476;
   1:L PR[91] R[100]mm/sec CNT100;
   1:  PR[91,1] = PR[90,1] + 49.408;
   1:  PR[91,2] = PR[90,2] + -10.911;
   1:L PR[91] R[100]mm/sec CNT100;
   1:  PR[91,1] = PR[90,1] + 51.186;
   1:  PR[91,2] = PR[90,2] + -12.768;
   1:L PR[91] R[100]mm/sec CNT100;
   1:  PR[91,1] = PR[90,1] + 52.835;
   1:  PR[91,2] = PR[90,2] + -14.684;
   1:L PR[91] R[100]mm/sec CNT100;
   1:  PR[91,1] = PR[90,1] + 53.211;
   1:  PR[91,2] = PR[90,2] + -14.985;
   1:L PR[91] R[100]mm/sec CNT100;
   1:  PR[91,1] = PR[90,1] + 56.860;
   1:  PR[91,2] = PR[90,2] + -17.522;
   1:L PR[91] R[100]mm/sec CNT100;
   1:  PR[91,1] = PR[90,1] + 58.877;
   1:  PR[91,2] = PR[90,2] + -18.500;
   1:L PR[91] R[100]mm/sec CNT100;
   1:  PR[91,1] = PR[90,1] + 61.208;
   1:  PR[91,2] = PR[90,2] + -19.410;
   1:L PR[91] R[100]mm/sec CNT100;
   1:  PR[91,1] = PR[90,1] + 64.943;
   1:  PR[91,2] = PR[90,2] + -20.322;
   1:L PR[91] R[100]mm/sec CNT100;
   1:  PR[91,1] = PR[90,1] + 65.668;
   1:  PR[91,2] = PR[90,2] + -20.430;
   1:L PR[91] R[100]mm/sec CNT100;
   1:  PR[91,1] = PR[90,1] + 68.583;
   1:  PR[91,2] = PR[90,2] + -20.534;
   1:L PR[91] R[100]mm/sec CNT100;
   1:  PR[91,1] = PR[90,1] + 70.360;
   1:  PR[91,2] = PR[90,2] + -20.634;
   1:L PR[91] R[100]mm/sec CNT100;
   1:  PR[91,1] = PR[90,1] + 74.988;
   1:  PR[91,2] = PR[90,2] + -19.914;
   1:L PR[91] R[100]mm/sec CNT100;
   1:  PR[91,1] = PR[90,1] + 76.141;
   1:  PR[91,2] = PR[90,2] + -19.489;
   1:L PR[91] R[100]mm/sec CNT100;
   1:  PR[91,1] = PR[90,1] + 79.280;
   1:  PR[91,2] = PR[90,2] + -18.285;
   1:L PR[91] R[100]mm/sec CNT100;
   1:  PR[91,1] = PR[90,1] + 80.968;
   1:  PR[91,2] = PR[90,2] + -17.210;
   1:L PR[91] R[100]mm/sec CNT100;
   1:  PR[91,1] = PR[90,1] + 83.067;
   1:  PR[91,2] = PR[90,2] + -15.837;
   1:L PR[91] R[100]mm/sec CNT100;
   1:  PR[91,1] = PR[90,1] + 84.877;
   1:  PR[91,2] = PR[90,2] + -14.031;
   1:L PR[91] R[100]mm/sec CNT100;
   1:  PR[91,1] = PR[90,1] + 86.185;
   1:  PR[91,2] = PR[90,2] + -12.701;
   1:L PR[91] R[100]mm/sec CNT100;
   1:  PR[91,1] = PR[90,1] + 88.511;
   1:  PR[91,2] = PR[90,2] + -9.016;
   1:L PR[91] R[100]mm/sec CNT100;
   1:  PR[91,1] = PR[90,1] + 89.942;
   1:  PR[91,2] = PR[90,2] + -4.965;
   1:L PR[91] R[100]mm/sec CNT100;
   1:  PR[91,1] = PR[90,1] + 90.431;
   1:  PR[91,2] = PR[90,2] + -0.729;
   1:L PR[91] R[100]mm/sec CNT100;
   1:  PR[91,1] = PR[90,1] + 89.942;
   1:  PR[91,2] = PR[90,2] + 3.506;
   1:L PR[91] R[100]mm/sec CNT100;
   1:  PR[91,1] = PR[90,1] + 88.511;
   1:  PR[91,2] = PR[90,2] + 7.557;
   1:L PR[91] R[100]mm/sec CNT100;
   1:  PR[91,1] = PR[90,1] + 86.191;
   1:  PR[91,2] = PR[90,2] + 11.233;
   1:L PR[91] R[100]mm/sec CNT100;
   1:  PR[91,1] = PR[90,1] + 84.368;
   1:  PR[91,2] = PR[90,2] + 13.048;
   1:L PR[91] R[100]mm/sec CNT100;
   1:  PR[91,1] = PR[90,1] + 83.067;
   1:  PR[91,2] = PR[90,2] + 14.375;
   1:L PR[91] R[100]mm/sec CNT100;
   1:  PR[91,1] = PR[90,1] + 81.258;
   1:  PR[91,2] = PR[90,2] + 15.525;
   1:L PR[91] R[100]mm/sec CNT100;
   1:  PR[91,1] = PR[90,1] + 79.280;
   1:  PR[91,2] = PR[90,2] + 16.823;
   1:L PR[91] R[100]mm/sec CNT100;
   1:  PR[91,1] = PR[90,1] + 77.780;
   1:  PR[91,2] = PR[90,2] + 17.372;
   1:L PR[91] R[100]mm/sec CNT100;
   1:  PR[91,1] = PR[90,1] + 74.987;
   1:  PR[91,2] = PR[90,2] + 18.452;
   1:L PR[91] R[100]mm/sec CNT100;
   1:  PR[91,1] = PR[90,1] + 74.070;
   1:  PR[91,2] = PR[90,2] + 18.580;
   1:L PR[91] R[100]mm/sec CNT100;
   1:  PR[91,1] = PR[90,1] + 70.356;
   1:  PR[91,2] = PR[90,2] + 19.175;
   1:L PR[91] R[100]mm/sec CNT100;
   1:  PR[91,1] = PR[90,1] + 68.583;
   1:  PR[91,2] = PR[90,2] + 19.075;
   1:L PR[91] R[100]mm/sec CNT100;
   1:  PR[91,1] = PR[90,1] + 65.668;
   1:  PR[91,2] = PR[90,2] + 18.971;
   1:L PR[91] R[100]mm/sec CNT100;
   1:  PR[91,1] = PR[90,1] + 64.944;
   1:  PR[91,2] = PR[90,2] + 18.863;
   1:L PR[91] R[100]mm/sec CNT100;
   1:  PR[91,1] = PR[90,1] + 61.208;
   1:  PR[91,2] = PR[90,2] + 17.952;
   1:L PR[91] R[100]mm/sec CNT100;
   1:  PR[91,1] = PR[90,1] + 58.878;
   1:  PR[91,2] = PR[90,2] + 17.042;
   1:L PR[91] R[100]mm/sec CNT100;
   1:  PR[91,1] = PR[90,1] + 56.860;
   1:  PR[91,2] = PR[90,2] + 16.064;
   1:L PR[91] R[100]mm/sec CNT100;
   1:  PR[91,1] = PR[90,1] + 53.212;
   1:  PR[91,2] = PR[90,2] + 13.527;
   1:L PR[91] R[100]mm/sec CNT100;
   1:  PR[91,1] = PR[90,1] + 52.836;
   1:  PR[91,2] = PR[90,2] + 13.226;
   1:L PR[91] R[100]mm/sec CNT100;
   1:  PR[91,1] = PR[90,1] + 51.186;
   1:  PR[91,2] = PR[90,2] + 11.309;
   1:L PR[91] R[100]mm/sec CNT100;
   1:  PR[91,1] = PR[90,1] + 49.400;
   1:  PR[91,2] = PR[90,2] + 9.445;
   1:L PR[91] R[100]mm/sec CNT100;
   1:  PR[91,1] = PR[90,1] + 49.055;
   1:  PR[91,2] = PR[90,2] + 9.026;
   1:L PR[91] R[100]mm/sec CNT100;
   1:  PR[91,1] = PR[90,1] + 47.153;
   1:  PR[91,2] = PR[90,2] + 5.377;
   1:L PR[91] R[100]mm/sec CNT100;
   1:  PR[91,1] = PR[90,1] + 45.494;
   1:  PR[91,2] = PR[90,2] + -0.780;
   1:L PR[91] R[100]mm/sec CNT100TB   .50sec,CALL END_PUD;
   1:  PR[92] = PR[91];
   1:  PR[92,3] = PR[92,3] + 20;
   1:J PR[92] 10% FINE;
   1:  PR[91,1] = PR[90,1] + -2.545;
   1:  PR[91,2] = PR[90,2] + -5.813;
   1:  PR[92] = PR[91];
   1:  PR[92,3] = PR[92,3] + 20;
   1:J PR[92] 10% FINE;
   1:L PR[91] R[100]mm/sec CNT100;
   1:  CALL LASER_DRAHT_START;
   1:  PR[91,1] = PR[90,1] + -2.063;
   1:  PR[91,2] = PR[90,2] + -3.251;
   1:L PR[91] R[100]mm/sec CNT100;
   1:  PR[91,1] = PR[90,1] + -1.845;
   1:  PR[91,2] = PR[90,2] + -1.444;
   1:L PR[91] R[100]mm/sec CNT100;
   1:  PR[91,1] = PR[90,1] + -1.827;
   1:  PR[91,2] = PR[90,2] + -0.821;
   1:L PR[91] R[100]mm/sec CNT100;
   1:  PR[91,1] = PR[90,1] + -2.052;
   1:  PR[91,2] = PR[90,2] + 1.043;
   1:L PR[91] R[100]mm/sec CNT100;
   1:  PR[91,1] = PR[90,1] + -2.079;
   1:  PR[91,2] = PR[90,2] + 1.870;
   1:L PR[91] R[100]mm/sec CNT100;
   1:  PR[91,1] = PR[90,1] + -2.542;
   1:  PR[91,2] = PR[90,2] + 4.345;
   1:L PR[91] R[100]mm/sec CNT100;
   1:  PR[91,1] = PR[90,1] + -3.216;
   1:  PR[91,2] = PR[90,2] + 6.152;
   1:L PR[91] R[100]mm/sec CNT100;
   1:  PR[91,1] = PR[90,1] + -4.219;
   1:  PR[91,2] = PR[90,2] + 8.369;
   1:L PR[91] R[100]mm/sec CNT100;
   1:  PR[91,1] = PR[90,1] + -5.449;
   1:  PR[91,2] = PR[90,2] + 10.199;
   1:L PR[91] R[100]mm/sec CNT100;
   1:  PR[91,1] = PR[90,1] + -6.767;
   1:  PR[91,2] = PR[90,2] + 11.903;
   1:L PR[91] R[100]mm/sec CNT100;
   1:  PR[91,1] = PR[90,1] + -8.663;
   1:  PR[91,2] = PR[90,2] + 13.664;
   1:L PR[91] R[100]mm/sec CNT100;
   1:  PR[91,1] = PR[90,1] + -10.039;
   1:  PR[91,2] = PR[90,2] + 14.785;
   1:L PR[91] R[100]mm/sec CNT100;
   1:  PR[91,1] = PR[90,1] + -12.675;
   1:  PR[91,2] = PR[90,2] + 16.303;
   1:L PR[91] R[100]mm/sec CNT100;
   1:  PR[91,1] = PR[90,1] + -13.864;
   1:  PR[91,2] = PR[90,2] + 16.892;
   1:L PR[91] R[100]mm/sec CNT100;
   1:  PR[91,1] = PR[90,1] + -17.226;
   1:  PR[91,2] = PR[90,2] + 17.935;
   1:L PR[91] R[100]mm/sec CNT100;
   1:  PR[91,1] = PR[90,1] + -18.054;
   1:  PR[91,2] = PR[90,2] + 18.138;
   1:L PR[91] R[100]mm/sec CNT100;
   1:  PR[91,1] = PR[90,1] + -22.027;
   1:  PR[91,2] = PR[90,2] + 18.466;
   1:L PR[91] R[100]mm/sec CNT100;
   1:  PR[91,1] = PR[90,1] + -22.408;
   1:  PR[91,2] = PR[90,2] + 18.476;
   1:L PR[91] R[100]mm/sec CNT100;
   1:  PR[91,1] = PR[90,1] + -26.777;
   1:  PR[91,2] = PR[90,2] + 17.875;
   1:L PR[91] R[100]mm/sec CNT100;
   1:  PR[91,1] = PR[90,1] + -30.837;
   1:  PR[91,2] = PR[90,2] + 16.394;
   1:L PR[91] R[100]mm/sec CNT100;
   1:  PR[91,1] = PR[90,1] + -34.445;
   1:  PR[91,2] = PR[90,2] + 14.080;
   1:L PR[91] R[100]mm/sec CNT100;
   1:  PR[91,1] = PR[90,1] + -37.440;
   1:  PR[91,2] = PR[90,2] + 11.049;
   1:L PR[91] R[100]mm/sec CNT100;
   1:  PR[91,1] = PR[90,1] + -39.685;
   1:  PR[91,2] = PR[90,2] + 7.452;
   1:L PR[91] R[100]mm/sec CNT100;
   1:  PR[91,1] = PR[90,1] + -41.074;
   1:  PR[91,2] = PR[90,2] + 3.459;
   1:L PR[91] R[100]mm/sec CNT100;
   1:  PR[91,1] = PR[90,1] + -41.552;
   1:  PR[91,2] = PR[90,2] + -0.720;
   1:L PR[91] R[100]mm/sec CNT100;
   1:  PR[91,1] = PR[90,1] + -41.468;
   1:  PR[91,2] = PR[90,2] + -1.394;
   1:L PR[91] R[100]mm/sec CNT100;
   1:  PR[91,1] = PR[90,1] + -41.073;
   1:  PR[91,2] = PR[90,2] + -4.920;
   1:L PR[91] R[100]mm/sec CNT100;
   1:  PR[91,1] = PR[90,1] + -39.685;
   1:  PR[91,2] = PR[90,2] + -8.910;
   1:L PR[91] R[100]mm/sec CNT100;
   1:  PR[91,1] = PR[90,1] + -37.440;
   1:  PR[91,2] = PR[90,2] + -12.508;
   1:L PR[91] R[100]mm/sec CNT100;
   1:  PR[91,1] = PR[90,1] + -34.445;
   1:  PR[91,2] = PR[90,2] + -15.539;
   1:L PR[91] R[100]mm/sec CNT100;
   1:  PR[91,1] = PR[90,1] + -30.837;
   1:  PR[91,2] = PR[90,2] + -17.853;
   1:L PR[91] R[100]mm/sec CNT100;
   1:  PR[91,1] = PR[90,1] + -26.738;
   1:  PR[91,2] = PR[90,2] + -19.348;
   1:L PR[91] R[100]mm/sec CNT100;
   1:  PR[91,1] = PR[90,1] + -22.411;
   1:  PR[91,2] = PR[90,2] + -19.935;
   1:L PR[91] R[100]mm/sec CNT100;
   1:  PR[91,1] = PR[90,1] + -22.029;
   1:  PR[91,2] = PR[90,2] + -19.925;
   1:L PR[91] R[100]mm/sec CNT100;
   1:  PR[91,1] = PR[90,1] + -18.057;
   1:  PR[91,2] = PR[90,2] + -19.597;
   1:L PR[91] R[100]mm/sec CNT100;
   1:  PR[91,1] = PR[90,1] + -17.229;
   1:  PR[91,2] = PR[90,2] + -19.395;
   1:L PR[91] R[100]mm/sec CNT100;
   1:  PR[91,1] = PR[90,1] + -13.868;
   1:  PR[91,2] = PR[90,2] + -18.353;
   1:L PR[91] R[100]mm/sec CNT100;
   1:  PR[91,1] = PR[90,1] + -12.679;
   1:  PR[91,2] = PR[90,2] + -17.764;
   1:L PR[91] R[100]mm/sec CNT100;
   1:  PR[91,1] = PR[90,1] + -10.044;
   1:  PR[91,2] = PR[90,2] + -16.246;
   1:L PR[91] R[100]mm/sec CNT100;
   1:  PR[91,1] = PR[90,1] + -8.668;
   1:  PR[91,2] = PR[90,2] + -15.128;
   1:L PR[91] R[100]mm/sec CNT100;
   1:  PR[91,1] = PR[90,1] + -6.772;
   1:  PR[91,2] = PR[90,2] + -13.367;
   1:L PR[91] R[100]mm/sec CNT100;
   1:  PR[91,1] = PR[90,1] + -5.454;
   1:  PR[91,2] = PR[90,2] + -11.665;
   1:L PR[91] R[100]mm/sec CNT100;
   1:  PR[91,1] = PR[90,1] + -4.223;
   1:  PR[91,2] = PR[90,2] + -9.835;
   1:L PR[91] R[100]mm/sec CNT100;
   1:  PR[91,1] = PR[90,1] + -3.219;
   1:  PR[91,2] = PR[90,2] + -7.620;
   1:L PR[91] R[100]mm/sec CNT100;
   1:  PR[91,1] = PR[90,1] + -2.545;
   1:  PR[91,2] = PR[90,2] + -5.813;
   1:L PR[91] R[100]mm/sec CNT100TB   .50sec,CALL END_PUD;
   1:  PR[92] = PR[91];
   1:  PR[92,3] = PR[92,3] + 20;
   1:J PR[92] 10% FINE;
   1:  PR[91,1] = PR[90,1] + -49.402;
   1:  PR[91,2] = PR[90,2] + 2.907;
   1:  PR[92] = PR[91];
   1:  PR[92,3] = PR[92,3] + 20;
   1:J PR[92] 10% FINE;
   1:L PR[91] R[100]mm/sec CNT100;
   1:  CALL LASER_DRAHT_START;
   1:  PR[91,1] = PR[90,1] + -49.455;
   1:  PR[91,2] = PR[90,2] + 3.404;
   1:L PR[91] R[100]mm/sec CNT100;
   1:  PR[91,1] = PR[90,1] + -50.286;
   1:  PR[91,2] = PR[90,2] + 5.455;
   1:L PR[91] R[100]mm/sec CNT100;
   1:  PR[91,1] = PR[90,1] + -50.999;
   1:  PR[91,2] = PR[90,2] + 7.343;
   1:L PR[91] R[100]mm/sec CNT100;
   1:  PR[91,1] = PR[90,1] + -53.381;
   1:  PR[91,2] = PR[90,2] + 10.875;
   1:L PR[91] R[100]mm/sec CNT100;
   1:  PR[91,1] = PR[90,1] + -56.525;
   1:  PR[91,2] = PR[90,2] + 13.850;
   1:L PR[91] R[100]mm/sec CNT100;
   1:  PR[91,1] = PR[90,1] + -58.321;
   1:  PR[91,2] = PR[90,2] + 14.961;
   1:L PR[91] R[100]mm/sec CNT100;
   1:  PR[91,1] = PR[90,1] + -60.248;
   1:  PR[91,2] = PR[90,2] + 16.125;
   1:L PR[91] R[100]mm/sec CNT100;
   1:  PR[91,1] = PR[90,1] + -64.390;
   1:  PR[91,2] = PR[90,2] + 17.634;
   1:L PR[91] R[100]mm/sec CNT100;
   1:  PR[91,1] = PR[90,1] + -68.740;
   1:  PR[91,2] = PR[90,2] + 18.318;
   1:L PR[91] R[100]mm/sec CNT100;
   1:  PR[91,1] = PR[90,1] + -72.934;
   1:  PR[91,2] = PR[90,2] + 18.197;
   1:L PR[91] R[100]mm/sec CNT100;
   1:  PR[91,1] = PR[90,1] + -76.974;
   1:  PR[91,2] = PR[90,2] + 17.263;
   1:L PR[91] R[100]mm/sec CNT100;
   1:  PR[91,1] = PR[90,1] + -80.705;
   1:  PR[91,2] = PR[90,2] + 15.568;
   1:L PR[91] R[100]mm/sec CNT100;
   1:  PR[91,1] = PR[90,1] + -83.979;
   1:  PR[91,2] = PR[90,2] + 13.192;
   1:L PR[91] R[100]mm/sec CNT100;
   1:  PR[91,1] = PR[90,1] + -86.664;
   1:  PR[91,2] = PR[90,2] + 10.240;
   1:L PR[91] R[100]mm/sec CNT100;
   1:  PR[91,1] = PR[90,1] + -88.659;
   1:  PR[91,2] = PR[90,2] + 6.841;
   1:L PR[91] R[100]mm/sec CNT100;
   1:  PR[91,1] = PR[90,1] + -89.885;
   1:  PR[91,2] = PR[90,2] + 3.132;
   1:L PR[91] R[100]mm/sec CNT100;
   1:  PR[91,1] = PR[90,1] + -90.196;
   1:  PR[91,2] = PR[90,2] + 0.271;
   1:L PR[91] R[100]mm/sec CNT100;
   1:  PR[91,1] = PR[90,1] + -90.379;
   1:  PR[91,2] = PR[90,2] + -0.638;
   1:L PR[91] R[100]mm/sec CNT100;
   1:  PR[91,1] = PR[90,1] + -90.388;
   1:  PR[91,2] = PR[90,2] + -0.728;
   1:L PR[91] R[100]mm/sec CNT100;
   1:  PR[91,1] = PR[90,1] + -90.009;
   1:  PR[91,2] = PR[90,2] + -4.217;
   1:L PR[91] R[100]mm/sec CNT100;
   1:  PR[91,1] = PR[90,1] + -89.978;
   1:  PR[91,2] = PR[90,2] + -4.355;
   1:L PR[91] R[100]mm/sec CNT100;
   1:  PR[91,1] = PR[90,1] + -89.953;
   1:  PR[91,2] = PR[90,2] + -4.588;
   1:L PR[91] R[100]mm/sec CNT100;
   1:  PR[91,1] = PR[90,1] + -88.720;
   1:  PR[91,2] = PR[90,2] + -8.290;
   1:L PR[91] R[100]mm/sec CNT100;
   1:  PR[91,1] = PR[90,1] + -86.710;
   1:  PR[91,2] = PR[90,2] + -11.689;
   1:L PR[91] R[100]mm/sec CNT100;
   1:  PR[91,1] = PR[90,1] + -84.003;
   1:  PR[91,2] = PR[90,2] + -14.643;
   1:L PR[91] R[100]mm/sec CNT100;
   1:  PR[91,1] = PR[90,1] + -80.703;
   1:  PR[91,2] = PR[90,2] + -17.023;
   1:L PR[91] R[100]mm/sec CNT100;
   1:  PR[91,1] = PR[90,1] + -78.294;
   1:  PR[91,2] = PR[90,2] + -18.099;
   1:L PR[91] R[100]mm/sec CNT100;
   1:  PR[91,1] = PR[90,1] + -76.929;
   1:  PR[91,2] = PR[90,2] + -18.728;
   1:L PR[91] R[100]mm/sec CNT100;
   1:  PR[91,1] = PR[90,1] + -74.807;
   1:  PR[91,2] = PR[90,2] + -19.203;
   1:L PR[91] R[100]mm/sec CNT100;
   1:  PR[91,1] = PR[90,1] + -72.849;
   1:  PR[91,2] = PR[90,2] + -19.670;
   1:L PR[91] R[100]mm/sec CNT100;
   1:  PR[91,1] = PR[90,1] + -71.213;
   1:  PR[91,2] = PR[90,2] + -19.706;
   1:L PR[91] R[100]mm/sec CNT100;
   1:  PR[91,1] = PR[90,1] + -68.622;
   1:  PR[91,2] = PR[90,2] + -19.800;
   1:L PR[91] R[100]mm/sec CNT100;
   1:  PR[91,1] = PR[90,1] + -67.618;
   1:  PR[91,2] = PR[90,2] + -19.621;
   1:L PR[91] R[100]mm/sec CNT100;
   1:  PR[91,1] = PR[90,1] + -64.414;
   1:  PR[91,2] = PR[90,2] + -19.098;
   1:L PR[91] R[100]mm/sec CNT100;
   1:  PR[91,1] = PR[90,1] + -61.199;
   1:  PR[91,2] = PR[90,2] + -17.867;
   1:L PR[91] R[100]mm/sec CNT100;
   1:  PR[91,1] = PR[90,1] + -60.331;
   1:  PR[91,2] = PR[90,2] + -17.562;
   1:L PR[91] R[100]mm/sec CNT100;
   1:  PR[91,1] = PR[90,1] + -57.147;
   1:  PR[91,2] = PR[90,2] + -15.650;
   1:L PR[91] R[100]mm/sec CNT100;
   1:  PR[91,1] = PR[90,1] + -56.507;
   1:  PR[91,2] = PR[90,2] + -15.281;
   1:L PR[91] R[100]mm/sec CNT100;
   1:  PR[91,1] = PR[90,1] + -54.384;
   1:  PR[91,2] = PR[90,2] + -13.299;
   1:L PR[91] R[100]mm/sec CNT100;
   1:  PR[91,1] = PR[90,1] + -53.299;
   1:  PR[91,2] = PR[90,2] + -12.318;
   1:L PR[91] R[100]mm/sec CNT100;
   1:  PR[91,1] = PR[90,1] + -52.069;
   1:  PR[91,2] = PR[90,2] + -10.516;
   1:L PR[91] R[100]mm/sec CNT100;
   1:  PR[91,1] = PR[90,1] + -50.858;
   1:  PR[91,2] = PR[90,2] + -8.788;
   1:L PR[91] R[100]mm/sec CNT100;
   1:  PR[91,1] = PR[90,1] + -49.338;
   1:  PR[91,2] = PR[90,2] + -4.866;
   1:L PR[91] R[100]mm/sec CNT100;
   1:  PR[91,1] = PR[90,1] + -49.195;
   1:  PR[91,2] = PR[90,2] + -3.713;
   1:L PR[91] R[100]mm/sec CNT100;
   1:  PR[91,1] = PR[90,1] + -49.053;
   1:  PR[91,2] = PR[90,2] + -1.681;
   1:L PR[91] R[100]mm/sec CNT100;
   1:  PR[91,1] = PR[90,1] + -48.931;
   1:  PR[91,2] = PR[90,2] + -0.731;
   1:L PR[91] R[100]mm/sec CNT100;
   1:  PR[91,1] = PR[90,1] + -49.402;
   1:  PR[91,2] = PR[90,2] + 2.907;
   1:L PR[91] R[100]mm/sec CNT100TB   .50sec,CALL END_PUD;
   1:  PR[92] = PR[91];
   1:  PR[92,3] = PR[92,3] + 20;
   1:J PR[92] 10% FINE;
   1:  PR[91] = PR[90];
   1:  PR[91,1] = PR[90,1] + 69.952;
   1:  PR[91,2] = PR[90,2] + 19.345;
   1:  PR[91,3] = PR[90,3] + 35.295;
   1:  PR[92] = PR[91];
   1:  PR[92,3] = PR[92,3] + 20;
   1:J PR[92] 10% FINE;
   1:L PR[91] R[100]mm/sec CNT100;
   1:  CALL LASER_DRAHT_START;
   1:  PR[91,1] = PR[90,1] + 69.657;
   1:  PR[91,2] = PR[90,2] + 19.366;
   1:L PR[91] R[100]mm/sec CNT100;
   1:  PR[91,1] = PR[90,1] + 65.452;
   1:  PR[91,2] = PR[90,2] + 19.215;
   1:L PR[91] R[100]mm/sec CNT100;
   1:  PR[91,1] = PR[90,1] + 63.586;
   1:  PR[91,2] = PR[90,2] + 18.937;
   1:L PR[91] R[100]mm/sec CNT100;
   1:  PR[91,1] = PR[90,1] + 60.886;
   1:  PR[91,2] = PR[90,2] + 18.279;
   1:L PR[91] R[100]mm/sec CNT100;
   1:  PR[91,1] = PR[90,1] + 57.334;
   1:  PR[91,2] = PR[90,2] + 16.892;
   1:L PR[91] R[100]mm/sec CNT100;
   1:  PR[91,1] = PR[90,1] + 56.403;
   1:  PR[91,2] = PR[90,2] + 16.440;
   1:L PR[91] R[100]mm/sec CNT100;
   1:  PR[91,1] = PR[90,1] + 53.336;
   1:  PR[91,2] = PR[90,2] + 14.308;
   1:L PR[91] R[100]mm/sec CNT100;
   1:  PR[91,1] = PR[90,1] + 52.055;
   1:  PR[91,2] = PR[90,2] + 13.518;
   1:L PR[91] R[100]mm/sec CNT100;
   1:  PR[91,1] = PR[90,1] + 51.768;
   1:  PR[91,2] = PR[90,2] + 13.306;
   1:L PR[91] R[100]mm/sec CNT100;
   1:  PR[91,1] = PR[90,1] + 48.909;
   1:  PR[91,2] = PR[90,2] + 10.322;
   1:L PR[91] R[100]mm/sec CNT100;
   1:  PR[91,1] = PR[90,1] + 47.681;
   1:  PR[91,2] = PR[90,2] + 8.831;
   1:L PR[91] R[100]mm/sec CNT100;
   1:  PR[91,1] = PR[90,1] + 46.544;
   1:  PR[91,2] = PR[90,2] + 6.639;
   1:L PR[91] R[100]mm/sec CNT100;
   1:  PR[91,1] = PR[90,1] + 44.305;
   1:  PR[91,2] = PR[90,2] + 2.562;
   1:L PR[91] R[100]mm/sec CNT100;
   1:  PR[91,1] = PR[90,1] + 41.592;
   1:  PR[91,2] = PR[90,2] + 8.703;
   1:L PR[91] R[100]mm/sec CNT100;
   1:  PR[91,1] = PR[90,1] + 41.274;
   1:  PR[91,2] = PR[90,2] + 9.287;
   1:L PR[91] R[100]mm/sec CNT100;
   1:  PR[91,1] = PR[90,1] + 40.590;
   1:  PR[91,2] = PR[90,2] + 10.194;
   1:L PR[91] R[100]mm/sec CNT100;
   1:  PR[91,1] = PR[90,1] + 38.016;
   1:  PR[91,2] = PR[90,2] + 13.467;
   1:L PR[91] R[100]mm/sec CNT100;
   1:  PR[91,1] = PR[90,1] + 37.291;
   1:  PR[91,2] = PR[90,2] + 14.026;
   1:L PR[91] R[100]mm/sec CNT100;
   1:  PR[91,1] = PR[90,1] + 33.908;
   1:  PR[91,2] = PR[90,2] + 16.575;
   1:L PR[91] R[100]mm/sec CNT100;
   1:  PR[91,1] = PR[90,1] + 29.117;
   1:  PR[91,2] = PR[90,2] + 18.537;
   1:L PR[91] R[100]mm/sec CNT100;
   1:  PR[91,1] = PR[90,1] + 28.399;
   1:  PR[91,2] = PR[90,2] + 18.634;
   1:L PR[91] R[100]mm/sec CNT100;
   1:  PR[91,1] = PR[90,1] + 23.987;
   1:  PR[91,2] = PR[90,2] + 19.202;
   1:L PR[91] R[100]mm/sec CNT100;
   1:  PR[91,1] = PR[90,1] + 18.842;
   1:  PR[91,2] = PR[90,2] + 18.522;
   1:L PR[91] R[100]mm/sec CNT100;
   1:  PR[91,1] = PR[90,1] + 14.039;
   1:  PR[91,2] = PR[90,2] + 16.538;
   1:L PR[91] R[100]mm/sec CNT100;
   1:  PR[91,1] = PR[90,1] + 9.906;
   1:  PR[91,2] = PR[90,2] + 13.378;
   1:L PR[91] R[100]mm/sec CNT100;
   1:  PR[91,1] = PR[90,1] + 6.730;
   1:  PR[91,2] = PR[90,2] + 9.250;
   1:L PR[91] R[100]mm/sec CNT100;
   1:  PR[91,1] = PR[90,1] + 4.730;
   1:  PR[91,2] = PR[90,2] + 4.439;
   1:L PR[91] R[100]mm/sec CNT100;
   1:  PR[91,1] = PR[90,1] + 4.049;
   1:  PR[91,2] = PR[90,2] + -0.729;
   1:L PR[91] R[100]mm/sec CNT100;
   1:  PR[91,1] = PR[90,1] + 4.732;
   1:  PR[91,2] = PR[90,2] + -5.902;
   1:L PR[91] R[100]mm/sec CNT100;
   1:  PR[91,1] = PR[90,1] + 6.735;
   1:  PR[91,2] = PR[90,2] + -10.718;
   1:L PR[91] R[100]mm/sec CNT100;
   1:  PR[91,1] = PR[90,1] + 9.916;
   1:  PR[91,2] = PR[90,2] + -14.847;
   1:L PR[91] R[100]mm/sec CNT100;
   1:  PR[91,1] = PR[90,1] + 14.056;
   1:  PR[91,2] = PR[90,2] + -18.006;
   1:L PR[91] R[100]mm/sec CNT100;
   1:  PR[91,1] = PR[90,1] + 18.865;
   1:  PR[91,2] = PR[90,2] + -19.987;
   1:L PR[91] R[100]mm/sec CNT100;
   1:  PR[91,1] = PR[90,1] + 24.014;
   1:  PR[91,2] = PR[90,2] + -20.661;
   1:L PR[91] R[100]mm/sec CNT100;
   1:  PR[91,1] = PR[90,1] + 28.429;
   1:  PR[91,2] = PR[90,2] + -20.085;
   1:L PR[91] R[100]mm/sec CNT100;
   1:  PR[91,1] = PR[90,1] + 29.148;
   1:  PR[91,2] = PR[90,2] + -19.987;
   1:L PR[91] R[100]mm/sec CNT100;
   1:  PR[91,1] = PR[90,1] + 33.936;
   1:  PR[91,2] = PR[90,2] + -18.017;
   1:L PR[91] R[100]mm/sec CNT100;
   1:  PR[91,1] = PR[90,1] + 38.048;
   1:  PR[91,2] = PR[90,2] + -14.892;
   1:L PR[91] R[100]mm/sec CNT100;
   1:  PR[91,1] = PR[90,1] + 40.630;
   1:  PR[91,2] = PR[90,2] + -11.589;
   1:L PR[91] R[100]mm/sec CNT100;
   1:  PR[91,1] = PR[90,1] + 41.273;
   1:  PR[91,2] = PR[90,2] + -10.747;
   1:L PR[91] R[100]mm/sec CNT100;
   1:  PR[91,1] = PR[90,1] + 41.543;
   1:  PR[91,2] = PR[90,2] + -10.255;
   1:L PR[91] R[100]mm/sec CNT100;
   1:  PR[91,1] = PR[90,1] + 41.867;
   1:  PR[91,2] = PR[90,2] + -9.470;
   1:L PR[91] R[100]mm/sec CNT100;
   1:  PR[91,1] = PR[90,1] + 44.364;
   1:  PR[91,2] = PR[90,2] + -3.909;
   1:L PR[91] R[100]mm/sec CNT100;
   1:  PR[91,1] = PR[90,1] + 47.704;
   1:  PR[91,2] = PR[90,2] + -10.331;
   1:L PR[91] R[100]mm/sec CNT100;
   1:  PR[91,1] = PR[90,1] + 48.926;
   1:  PR[91,2] = PR[90,2] + -11.795;
   1:L PR[91] R[100]mm/sec CNT100;
   1:  PR[91,1] = PR[90,1] + 51.775;
   1:  PR[91,2] = PR[90,2] + -14.772;
   1:L PR[91] R[100]mm/sec CNT100;
   1:  PR[91,1] = PR[90,1] + 52.056;
   1:  PR[91,2] = PR[90,2] + -14.978;
   1:L PR[91] R[100]mm/sec CNT100;
   1:  PR[91,1] = PR[90,1] + 53.337;
   1:  PR[91,2] = PR[90,2] + -15.767;
   1:L PR[91] R[100]mm/sec CNT100;
   1:  PR[91,1] = PR[90,1] + 56.402;
   1:  PR[91,2] = PR[90,2] + -17.898;
   1:L PR[91] R[100]mm/sec CNT100;
   1:  PR[91,1] = PR[90,1] + 57.333;
   1:  PR[91,2] = PR[90,2] + -18.350;
   1:L PR[91] R[100]mm/sec CNT100;
   1:  PR[91,1] = PR[90,1] + 60.886;
   1:  PR[91,2] = PR[90,2] + -19.737;
   1:L PR[91] R[100]mm/sec CNT100;
   1:  PR[91,1] = PR[90,1] + 63.586;
   1:  PR[91,2] = PR[90,2] + -20.396;
   1:L PR[91] R[100]mm/sec CNT100;
   1:  PR[91,1] = PR[90,1] + 65.452;
   1:  PR[91,2] = PR[90,2] + -20.674;
   1:L PR[91] R[100]mm/sec CNT100;
   1:  PR[91,1] = PR[90,1] + 69.656;
   1:  PR[91,2] = PR[90,2] + -20.825;
   1:L PR[91] R[100]mm/sec CNT100;
   1:  PR[91,1] = PR[90,1] + 69.952;
   1:  PR[91,2] = PR[90,2] + -20.804;
   1:L PR[91] R[100]mm/sec CNT100;
   1:  PR[91,1] = PR[90,1] + 71.659;
   1:  PR[91,2] = PR[90,2] + -20.520;
   1:L PR[91] R[100]mm/sec CNT100;
   1:  PR[91,1] = PR[90,1] + 74.623;
   1:  PR[91,2] = PR[90,2] + -20.055;
   1:L PR[91] R[100]mm/sec CNT100;
   1:  PR[91,1] = PR[90,1] + 75.033;
   1:  PR[91,2] = PR[90,2] + -19.903;
   1:L PR[91] R[100]mm/sec CNT100;
   1:  PR[91,1] = PR[90,1] + 78.943;
   1:  PR[91,2] = PR[90,2] + -18.404;
   1:L PR[91] R[100]mm/sec CNT100;
   1:  PR[91,1] = PR[90,1] + 80.020;
   1:  PR[91,2] = PR[90,2] + -17.717;
   1:L PR[91] R[100]mm/sec CNT100;
   1:  PR[91,1] = PR[90,1] + 82.749;
   1:  PR[91,2] = PR[90,2] + -15.933;
   1:L PR[91] R[100]mm/sec CNT100;
   1:  PR[91,1] = PR[90,1] + 84.089;
   1:  PR[91,2] = PR[90,2] + -14.597;
   1:L PR[91] R[100]mm/sec CNT100;
   1:  PR[91,1] = PR[90,1] + 85.881;
   1:  PR[91,2] = PR[90,2] + -12.773;
   1:L PR[91] R[100]mm/sec CNT100;
   1:  PR[91,1] = PR[90,1] + 88.217;
   1:  PR[91,2] = PR[90,2] + -9.066;
   1:L PR[91] R[100]mm/sec CNT100;
   1:  PR[91,1] = PR[90,1] + 89.654;
   1:  PR[91,2] = PR[90,2] + -4.990;
   1:L PR[91] R[100]mm/sec CNT100;
   1:  PR[91,1] = PR[90,1] + 90.143;
   1:  PR[91,2] = PR[90,2] + -0.729;
   1:L PR[91] R[100]mm/sec CNT100;
   1:  PR[91,1] = PR[90,1] + 89.654;
   1:  PR[91,2] = PR[90,2] + 3.531;
   1:L PR[91] R[100]mm/sec CNT100;
   1:  PR[91,1] = PR[90,1] + 88.218;
   1:  PR[91,2] = PR[90,2] + 7.603;
   1:L PR[91] R[100]mm/sec CNT100;
   1:  PR[91,1] = PR[90,1] + 86.960;
   1:  PR[91,2] = PR[90,2] + 9.583;
   1:L PR[91] R[100]mm/sec CNT100;
   1:  PR[91,1] = PR[90,1] + 85.883;
   1:  PR[91,2] = PR[90,2] + 11.309;
   1:L PR[91] R[100]mm/sec CNT100;
   1:  PR[91,1] = PR[90,1] + 84.452;
   1:  PR[91,2] = PR[90,2] + 12.734;
   1:L PR[91] R[100]mm/sec CNT100;
   1:  PR[91,1] = PR[90,1] + 82.749;
   1:  PR[91,2] = PR[90,2] + 14.471;
   1:L PR[91] R[100]mm/sec CNT100;
   1:  PR[91,1] = PR[90,1] + 81.417;
   1:  PR[91,2] = PR[90,2] + 15.317;
   1:L PR[91] R[100]mm/sec CNT100;
   1:  PR[91,1] = PR[90,1] + 78.943;
   1:  PR[91,2] = PR[90,2] + 16.942;
   1:L PR[91] R[100]mm/sec CNT100;
   1:  PR[91,1] = PR[90,1] + 77.998;
   1:  PR[91,2] = PR[90,2] + 17.288;
   1:L PR[91] R[100]mm/sec CNT100;
   1:  PR[91,1] = PR[90,1] + 74.607;
   1:  PR[91,2] = PR[90,2] + 18.598;
   1:L PR[91] R[100]mm/sec CNT100;
   1:  PR[91,1] = PR[90,1] + 71.659;
   1:  PR[91,2] = PR[90,2] + 19.061;
   1:L PR[91] R[100]mm/sec CNT100;
   1:  PR[91,1] = PR[90,1] + 69.952;
   1:  PR[91,2] = PR[90,2] + 19.345;
   1:L PR[91] R[100]mm/sec CNT100TB   .50sec,CALL END_PUD;
   1:  PR[92] = PR[91];
   1:  PR[92,3] = PR[92,3] + 20;
   1:J PR[92] 10% FINE;
   1:  PR[91,1] = PR[90,1] + -21.225;
   1:  PR[91,2] = PR[90,2] + -20.035;
   1:  PR[92] = PR[91];
   1:  PR[92,3] = PR[92,3] + 20;
   1:J PR[92] 10% FINE;
   1:L PR[91] R[100]mm/sec CNT100;
   1:  CALL LASER_DRAHT_START;
   1:  PR[91,1] = PR[90,1] + -17.834;
   1:  PR[91,2] = PR[90,2] + -19.755;
   1:L PR[91] R[100]mm/sec CNT100;
   1:  PR[91,1] = PR[90,1] + -16.393;
   1:  PR[91,2] = PR[90,2] + -19.403;
   1:L PR[91] R[100]mm/sec CNT100;
   1:  PR[91,1] = PR[90,1] + -13.614;
   1:  PR[91,2] = PR[90,2] + -18.541;
   1:L PR[91] R[100]mm/sec CNT100;
   1:  PR[91,1] = PR[90,1] + -11.836;
   1:  PR[91,2] = PR[90,2] + -17.662;
   1:L PR[91] R[100]mm/sec CNT100;
   1:  PR[91,1] = PR[90,1] + -9.749;
   1:  PR[91,2] = PR[90,2] + -16.459;
   1:L PR[91] R[100]mm/sec CNT100;
   1:  PR[91,1] = PR[90,1] + -7.849;
   1:  PR[91,2] = PR[90,2] + -14.914;
   1:L PR[91] R[100]mm/sec CNT100;
   1:  PR[91,1] = PR[90,1] + -6.429;
   1:  PR[91,2] = PR[90,2] + -13.596;
   1:L PR[91] R[100]mm/sec CNT100;
   1:  PR[91,1] = PR[90,1] + -4.688;
   1:  PR[91,2] = PR[90,2] + -11.349;
   1:L PR[91] R[100]mm/sec CNT100;
   1:  PR[91,1] = PR[90,1] + -3.827;
   1:  PR[91,2] = PR[90,2] + -10.067;
   1:L PR[91] R[100]mm/sec CNT100;
   1:  PR[91,1] = PR[90,1] + -2.535;
   1:  PR[91,2] = PR[90,2] + -7.218;
   1:L PR[91] R[100]mm/sec CNT100;
   1:  PR[91,1] = PR[90,1] + -2.094;
   1:  PR[91,2] = PR[90,2] + -6.035;
   1:L PR[91] R[100]mm/sec CNT100;
   1:  PR[91,1] = PR[90,1] + -1.483;
   1:  PR[91,2] = PR[90,2] + -2.786;
   1:L PR[91] R[100]mm/sec CNT100;
   1:  PR[91,1] = PR[90,1] + -1.346;
   1:  PR[91,2] = PR[90,2] + -1.651;
   1:L PR[91] R[100]mm/sec CNT100;
   1:  PR[91,1] = PR[90,1] + -1.323;
   1:  PR[91,2] = PR[90,2] + -0.821;
   1:L PR[91] R[100]mm/sec CNT100;
   1:  PR[91,1] = PR[90,1] + -1.464;
   1:  PR[91,2] = PR[90,2] + 0.357;
   1:L PR[91] R[100]mm/sec CNT100;
   1:  PR[91,1] = PR[90,1] + -1.499;
   1:  PR[91,2] = PR[90,2] + 1.403;
   1:L PR[91] R[100]mm/sec CNT100;
   1:  PR[91,1] = PR[90,1] + -2.091;
   1:  PR[91,2] = PR[90,2] + 4.565;
   1:L PR[91] R[100]mm/sec CNT100;
   1:  PR[91,1] = PR[90,1] + -2.532;
   1:  PR[91,2] = PR[90,2] + 5.748;
   1:L PR[91] R[100]mm/sec CNT100;
   1:  PR[91,1] = PR[90,1] + -3.821;
   1:  PR[91,2] = PR[90,2] + 8.599;
   1:L PR[91] R[100]mm/sec CNT100;
   1:  PR[91,1] = PR[90,1] + -4.683;
   1:  PR[91,2] = PR[90,2] + 9.880;
   1:L PR[91] R[100]mm/sec CNT100;
   1:  PR[91,1] = PR[90,1] + -6.422;
   1:  PR[91,2] = PR[90,2] + 12.130;
   1:L PR[91] R[100]mm/sec CNT100;
   1:  PR[91,1] = PR[90,1] + -7.842;
   1:  PR[91,2] = PR[90,2] + 13.448;
   1:L PR[91] R[100]mm/sec CNT100;
   1:  PR[91,1] = PR[90,1] + -9.742;
   1:  PR[91,2] = PR[90,2] + 14.996;
   1:L PR[91] R[100]mm/sec CNT100;
   1:  PR[91,1] = PR[90,1] + -11.830;
   1:  PR[91,2] = PR[90,2] + 16.199;
   1:L PR[91] R[100]mm/sec CNT100;
   1:  PR[91,1] = PR[90,1] + -13.608;
   1:  PR[91,2] = PR[90,2] + 17.080;
   1:L PR[91] R[100]mm/sec CNT100;
   1:  PR[91,1] = PR[90,1] + -16.388;
   1:  PR[91,2] = PR[90,2] + 17.942;
   1:L PR[91] R[100]mm/sec CNT100;
   1:  PR[91,1] = PR[90,1] + -17.830;
   1:  PR[91,2] = PR[90,2] + 18.295;
   1:L PR[91] R[100]mm/sec CNT100;
   1:  PR[91,1] = PR[90,1] + -21.221;
   1:  PR[91,2] = PR[90,2] + 18.576;
   1:L PR[91] R[100]mm/sec CNT100;
   1:  PR[91,1] = PR[90,1] + -22.208;
   1:  PR[91,2] = PR[90,2] + 18.600;
   1:L PR[91] R[100]mm/sec CNT100;
   1:  PR[91,1] = PR[90,1] + -26.020;
   1:  PR[91,2] = PR[90,2] + 18.084;
   1:L PR[91] R[100]mm/sec CNT100;
   1:  PR[91,1] = PR[90,1] + -26.539;
   1:  PR[91,2] = PR[90,2] + 17.984;
   1:L PR[91] R[100]mm/sec CNT100;
   1:  PR[91,1] = PR[90,1] + -30.506;
   1:  PR[91,2] = PR[90,2] + 16.533;
   1:L PR[91] R[100]mm/sec CNT100;
   1:  PR[91,1] = PR[90,1] + -30.622;
   1:  PR[91,2] = PR[90,2] + 16.484;
   1:L PR[91] R[100]mm/sec CNT100;
   1:  PR[91,1] = PR[90,1] + -34.299;
   1:  PR[91,2] = PR[90,2] + 14.135;
   1:L PR[91] R[100]mm/sec CNT100;
   1:  PR[91,1] = PR[90,1] + -37.304;
   1:  PR[91,2] = PR[90,2] + 11.094;
   1:L PR[91] R[100]mm/sec CNT100;
   1:  PR[91,1] = PR[90,1] + -39.555;
   1:  PR[91,2] = PR[90,2] + 7.482;
   1:L PR[91] R[100]mm/sec CNT100;
   1:  PR[91,1] = PR[90,1] + -40.947;
   1:  PR[91,2] = PR[90,2] + 3.475;
   1:L PR[91] R[100]mm/sec CNT100;
   1:  PR[91,1] = PR[90,1] + -41.422;
   1:  PR[91,2] = PR[90,2] + -0.718;
   1:L PR[91] R[100]mm/sec CNT100;
   1:  PR[91,1] = PR[90,1] + -41.389;
   1:  PR[91,2] = PR[90,2] + -0.982;
   1:L PR[91] R[100]mm/sec CNT100;
   1:  PR[91,1] = PR[90,1] + -40.947;
   1:  PR[91,2] = PR[90,2] + -4.935;
   1:L PR[91] R[100]mm/sec CNT100;
   1:  PR[91,1] = PR[90,1] + -39.555;
   1:  PR[91,2] = PR[90,2] + -8.940;
   1:L PR[91] R[100]mm/sec CNT100;
   1:  PR[91,1] = PR[90,1] + -37.304;
   1:  PR[91,2] = PR[90,2] + -12.552;
   1:L PR[91] R[100]mm/sec CNT100;
   1:  PR[91,1] = PR[90,1] + -34.300;
   1:  PR[91,2] = PR[90,2] + -15.594;
   1:L PR[91] R[100]mm/sec CNT100;
   1:  PR[91,1] = PR[90,1] + -30.622;
   1:  PR[91,2] = PR[90,2] + -17.943;
   1:L PR[91] R[100]mm/sec CNT100;
   1:  PR[91,1] = PR[90,1] + -30.507;
   1:  PR[91,2] = PR[90,2] + -17.992;
   1:L PR[91] R[100]mm/sec CNT100;
   1:  PR[91,1] = PR[90,1] + -26.540;
   1:  PR[91,2] = PR[90,2] + -19.442;
   1:L PR[91] R[100]mm/sec CNT100;
   1:  PR[91,1] = PR[90,1] + -26.022;
   1:  PR[91,2] = PR[90,2] + -19.543;
   1:L PR[91] R[100]mm/sec CNT100;
   1:  PR[91,1] = PR[90,1] + -22.211;
   1:  PR[91,2] = PR[90,2] + -20.059;
   1:L PR[91] R[100]mm/sec CNT100;
   1:  PR[91,1] = PR[90,1] + -21.225;
   1:  PR[91,2] = PR[90,2] + -20.035;
   1:L PR[91] R[100]mm/sec CNT100TB   .50sec,CALL END_PUD;
   1:  PR[92] = PR[91];
   1:  PR[92,3] = PR[92,3] + 20;
   1:J PR[92] 10% FINE;
   1:  PR[91,1] = PR[90,1] + -89.612;
   1:  PR[91,2] = PR[90,2] + -4.603;
   1:  PR[92] = PR[91];
   1:  PR[92,3] = PR[92,3] + 20;
   1:J PR[92] 10% FINE;
   1:L PR[91] R[100]mm/sec CNT100;
   1:  CALL LASER_DRAHT_START;
   1:  PR[91,1] = PR[90,1] + -88.374;
   1:  PR[91,2] = PR[90,2] + -8.320;
   1:L PR[91] R[100]mm/sec CNT100;
   1:  PR[91,1] = PR[90,1] + -86.359;
   1:  PR[91,2] = PR[90,2] + -11.734;
   1:L PR[91] R[100]mm/sec CNT100;
   1:  PR[91,1] = PR[90,1] + -83.646;
   1:  PR[91,2] = PR[90,2] + -14.700;
   1:L PR[91] R[100]mm/sec CNT100;
   1:  PR[91,1] = PR[90,1] + -81.589;
   1:  PR[91,2] = PR[90,2] + -16.174;
   1:L PR[91] R[100]mm/sec CNT100;
   1:  PR[91,1] = PR[90,1] + -80.327;
   1:  PR[91,2] = PR[90,2] + -17.098;
   1:L PR[91] R[100]mm/sec CNT100;
   1:  PR[91,1] = PR[90,1] + -78.378;
   1:  PR[91,2] = PR[90,2] + -17.969;
   1:L PR[91] R[100]mm/sec CNT100;
   1:  PR[91,1] = PR[90,1] + -76.545;
   1:  PR[91,2] = PR[90,2] + -18.813;
   1:L PR[91] R[100]mm/sec CNT100;
   1:  PR[91,1] = PR[90,1] + -74.930;
   1:  PR[91,2] = PR[90,2] + -19.175;
   1:L PR[91] R[100]mm/sec CNT100;
   1:  PR[91,1] = PR[90,1] + -72.446;
   1:  PR[91,2] = PR[90,2] + -19.767;
   1:L PR[91] R[100]mm/sec CNT100;
   1:  PR[91,1] = PR[90,1] + -71.357;
   1:  PR[91,2] = PR[90,2] + -19.791;
   1:L PR[91] R[100]mm/sec CNT100;
   1:  PR[91,1] = PR[90,1] + -68.183;
   1:  PR[91,2] = PR[90,2] + -19.907;
   1:L PR[91] R[100]mm/sec CNT100;
   1:  PR[91,1] = PR[90,1] + -63.917;
   1:  PR[91,2] = PR[90,2] + -19.209;
   1:L PR[91] R[100]mm/sec CNT100;
   1:  PR[91,1] = PR[90,1] + -60.270;
   1:  PR[91,2] = PR[90,2] + -17.914;
   1:L PR[91] R[100]mm/sec CNT100;
   1:  PR[91,1] = PR[90,1] + -59.627;
   1:  PR[91,2] = PR[90,2] + -17.699;
   1:L PR[91] R[100]mm/sec CNT100;
   1:  PR[91,1] = PR[90,1] + -57.061;
   1:  PR[91,2] = PR[90,2] + -16.158;
   1:L PR[91] R[100]mm/sec CNT100;
   1:  PR[91,1] = PR[90,1] + -55.776;
   1:  PR[91,2] = PR[90,2] + -15.417;
   1:L PR[91] R[100]mm/sec CNT100;
   1:  PR[91,1] = PR[90,1] + -54.204;
   1:  PR[91,2] = PR[90,2] + -13.950;
   1:L PR[91] R[100]mm/sec CNT100;
   1:  PR[91,1] = PR[90,1] + -52.527;
   1:  PR[91,2] = PR[90,2] + -12.434;
   1:L PR[91] R[100]mm/sec CNT100;
   1:  PR[91,1] = PR[90,1] + -51.753;
   1:  PR[91,2] = PR[90,2] + -11.300;
   1:L PR[91] R[100]mm/sec CNT100;
   1:  PR[91,1] = PR[90,1] + -50.050;
   1:  PR[91,2] = PR[90,2] + -8.871;
   1:L PR[91] R[100]mm/sec CNT100;
   1:  PR[91,1] = PR[90,1] + -48.508;
   1:  PR[91,2] = PR[90,2] + -4.909;
   1:L PR[91] R[100]mm/sec CNT100;
   1:  PR[91,1] = PR[90,1] + -48.480;
   1:  PR[91,2] = PR[90,2] + -4.681;
   1:L PR[91] R[100]mm/sec CNT100;
   1:  PR[91,1] = PR[90,1] + -48.428;
   1:  PR[91,2] = PR[90,2] + -3.939;
   1:L PR[91] R[100]mm/sec CNT100;
   1:  PR[91,1] = PR[90,1] + -48.016;
   1:  PR[91,2] = PR[90,2] + -0.731;
   1:L PR[91] R[100]mm/sec CNT100;
   1:  PR[91,1] = PR[90,1] + -48.104;
   1:  PR[91,2] = PR[90,2] + -0.048;
   1:L PR[91] R[100]mm/sec CNT100;
   1:  PR[91,1] = PR[90,1] + -48.291;
   1:  PR[91,2] = PR[90,2] + 2.128;
   1:L PR[91] R[100]mm/sec CNT100;
   1:  PR[91,1] = PR[90,1] + -48.464;
   1:  PR[91,2] = PR[90,2] + 3.428;
   1:L PR[91] R[100]mm/sec CNT100;
   1:  PR[91,1] = PR[90,1] + -50.071;
   1:  PR[91,2] = PR[90,2] + 7.381;
   1:L PR[91] R[100]mm/sec CNT100;
   1:  PR[91,1] = PR[90,1] + -52.667;
   1:  PR[91,2] = PR[90,2] + 10.955;
   1:L PR[91] R[100]mm/sec CNT100;
   1:  PR[91,1] = PR[90,1] + -55.865;
   1:  PR[91,2] = PR[90,2] + 13.968;
   1:L PR[91] R[100]mm/sec CNT100;
   1:  PR[91,1] = PR[90,1] + -59.639;
   1:  PR[91,2] = PR[90,2] + 16.261;
   1:L PR[91] R[100]mm/sec CNT100;
   1:  PR[91,1] = PR[90,1] + -61.792;
   1:  PR[91,2] = PR[90,2] + 17.051;
   1:L PR[91] R[100]mm/sec CNT100;
   1:  PR[91,1] = PR[90,1] + -63.801;
   1:  PR[91,2] = PR[90,2] + 17.766;
   1:L PR[91] R[100]mm/sec CNT100;
   1:  PR[91,1] = PR[90,1] + -68.191;
   1:  PR[91,2] = PR[90,2] + 18.444;
   1:L PR[91] R[100]mm/sec CNT100;
   1:  PR[91,1] = PR[90,1] + -72.567;
   1:  PR[91,2] = PR[90,2] + 18.287;
   1:L PR[91] R[100]mm/sec CNT100;
   1:  PR[91,1] = PR[90,1] + -76.629;
   1:  PR[91,2] = PR[90,2] + 17.342;
   1:L PR[91] R[100]mm/sec CNT100;
   1:  PR[91,1] = PR[90,1] + -80.374;
   1:  PR[91,2] = PR[90,2] + 15.635;
   1:L PR[91] R[100]mm/sec CNT100;
   1:  PR[91,1] = PR[90,1] + -83.658;
   1:  PR[91,2] = PR[90,2] + 13.247;
   1:L PR[91] R[100]mm/sec CNT100;
   1:  PR[91,1] = PR[90,1] + -86.351;
   1:  PR[91,2] = PR[90,2] + 10.282;
   1:L PR[91] R[100]mm/sec CNT100;
   1:  PR[91,1] = PR[90,1] + -88.351;
   1:  PR[91,2] = PR[90,2] + 6.868;
   1:L PR[91] R[100]mm/sec CNT100;
   1:  PR[91,1] = PR[90,1] + -89.581;
   1:  PR[91,2] = PR[90,2] + 3.146;
   1:L PR[91] R[100]mm/sec CNT100;
   1:  PR[91,1] = PR[90,1] + -89.835;
   1:  PR[91,2] = PR[90,2] + 0.801;
   1:L PR[91] R[100]mm/sec CNT100;
   1:  PR[91,1] = PR[90,1] + -89.986;
   1:  PR[91,2] = PR[90,2] + 0.050;
   1:L PR[91] R[100]mm/sec CNT100;
   1:  PR[91,1] = PR[90,1] + -90.069;
   1:  PR[91,2] = PR[90,2] + -0.728;
   1:L PR[91] R[100]mm/sec CNT100;
   1:  PR[91,1] = PR[90,1] + -89.760;
   1:  PR[91,2] = PR[90,2] + -3.570;
   1:L PR[91] R[100]mm/sec CNT100;
   1:  PR[91,1] = PR[90,1] + -89.687;
   1:  PR[91,2] = PR[90,2] + -3.899;
   1:L PR[91] R[100]mm/sec CNT100;
   1:  PR[91,1] = PR[90,1] + -89.612;
   1:  PR[91,2] = PR[90,2] + -4.603;
   1:L PR[91] R[100]mm/sec CNT100TB   .50sec,CALL END_PUD;
   1:  PR[92] = PR[91];
   1:  PR[92,3] = PR[92,3] + 20;
   1:J PR[92] 10% FINE;
   1:  PR[91] = PR[90];
   1:  PR[91,1] = PR[90,1] + 48.448;
   1:  PR[91,2] = PR[90,2] + -12.683;
   1:  PR[91,3] = PR[90,3] + 36.595;
   1:  PR[92] = PR[91];
   1:  PR[92,3] = PR[92,3] + 20;
   1:J PR[92] 10% FINE;
   1:L PR[91] R[100]mm/sec CNT100;
   1:  CALL LASER_DRAHT_START;
   1:  PR[91,1] = PR[90,1] + 50.330;
   1:  PR[91,2] = PR[90,2] + -14.650;
   1:L PR[91] R[100]mm/sec CNT100;
   1:  PR[91,1] = PR[90,1] + 51.696;
   1:  PR[91,2] = PR[90,2] + -15.650;
   1:L PR[91] R[100]mm/sec CNT100;
   1:  PR[91,1] = PR[90,1] + 55.883;
   1:  PR[91,2] = PR[90,2] + -18.236;
   1:L PR[91] R[100]mm/sec CNT100;
   1:  PR[91,1] = PR[90,1] + 60.564;
   1:  PR[91,2] = PR[90,2] + -20.064;
   1:L PR[91] R[100]mm/sec CNT100;
   1:  PR[91,1] = PR[90,1] + 62.228;
   1:  PR[91,2] = PR[90,2] + -20.470;
   1:L PR[91] R[100]mm/sec CNT100;
   1:  PR[91,1] = PR[90,1] + 65.235;
   1:  PR[91,2] = PR[90,2] + -20.918;
   1:L PR[91] R[100]mm/sec CNT100;
   1:  PR[91,1] = PR[90,1] + 68.507;
   1:  PR[91,2] = PR[90,2] + -21.035;
   1:L PR[91] R[100]mm/sec CNT100;
   1:  PR[91,1] = PR[90,1] + 69.807;
   1:  PR[91,2] = PR[90,2] + -20.945;
   1:L PR[91] R[100]mm/sec CNT100;
   1:  PR[91,1] = PR[90,1] + 74.194;
   1:  PR[91,2] = PR[90,2] + -20.214;
   1:L PR[91] R[100]mm/sec CNT100;
   1:  PR[91,1] = PR[90,1] + 78.605;
   1:  PR[91,2] = PR[90,2] + -18.523;
   1:L PR[91] R[100]mm/sec CNT100;
   1:  PR[91,1] = PR[90,1] + 79.073;
   1:  PR[91,2] = PR[90,2] + -18.225;
   1:L PR[91] R[100]mm/sec CNT100;
   1:  PR[91,1] = PR[90,1] + 82.426;
   1:  PR[91,2] = PR[90,2] + -16.033;
   1:L PR[91] R[100]mm/sec CNT100;
   1:  PR[91,1] = PR[90,1] + 85.579;
   1:  PR[91,2] = PR[90,2] + -12.844;
   1:L PR[91] R[100]mm/sec CNT100;
   1:  PR[91,1] = PR[90,1] + 87.923;
   1:  PR[91,2] = PR[90,2] + -9.115;
   1:L PR[91] R[100]mm/sec CNT100;
   1:  PR[91,1] = PR[90,1] + 89.365;
   1:  PR[91,2] = PR[90,2] + -5.015;
   1:L PR[91] R[100]mm/sec CNT100;
   1:  PR[91,1] = PR[90,1] + 89.856;
   1:  PR[91,2] = PR[90,2] + -0.729;
   1:L PR[91] R[100]mm/sec CNT100;
   1:  PR[91,1] = PR[90,1] + 89.365;
   1:  PR[91,2] = PR[90,2] + 3.556;
   1:L PR[91] R[100]mm/sec CNT100;
   1:  PR[91,1] = PR[90,1] + 87.924;
   1:  PR[91,2] = PR[90,2] + 7.651;
   1:L PR[91] R[100]mm/sec CNT100;
   1:  PR[91,1] = PR[90,1] + 86.953;
   1:  PR[91,2] = PR[90,2] + 9.179;
   1:L PR[91] R[100]mm/sec CNT100;
   1:  PR[91,1] = PR[90,1] + 85.580;
   1:  PR[91,2] = PR[90,2] + 11.381;
   1:L PR[91] R[100]mm/sec CNT100;
   1:  PR[91,1] = PR[90,1] + 84.536;
   1:  PR[91,2] = PR[90,2] + 12.421;
   1:L PR[91] R[100]mm/sec CNT100;
   1:  PR[91,1] = PR[90,1] + 82.432;
   1:  PR[91,2] = PR[90,2] + 14.567;
   1:L PR[91] R[100]mm/sec CNT100;
   1:  PR[91,1] = PR[90,1] + 81.577;
   1:  PR[91,2] = PR[90,2] + 15.110;
   1:L PR[91] R[100]mm/sec CNT100;
   1:  PR[91,1] = PR[90,1] + 78.593;
   1:  PR[91,2] = PR[90,2] + 17.069;
   1:L PR[91] R[100]mm/sec CNT100;
   1:  PR[91,1] = PR[90,1] + 74.194;
   1:  PR[91,2] = PR[90,2] + 18.755;
   1:L PR[91] R[100]mm/sec CNT100;
   1:  PR[91,1] = PR[90,1] + 69.807;
   1:  PR[91,2] = PR[90,2] + 19.486;
   1:L PR[91] R[100]mm/sec CNT100;
   1:  PR[91,1] = PR[90,1] + 68.508;
   1:  PR[91,2] = PR[90,2] + 19.576;
   1:L PR[91] R[100]mm/sec CNT100;
   1:  PR[91,1] = PR[90,1] + 65.236;
   1:  PR[91,2] = PR[90,2] + 19.459;
   1:L PR[91] R[100]mm/sec CNT100;
   1:  PR[91,1] = PR[90,1] + 62.229;
   1:  PR[91,2] = PR[90,2] + 19.012;
   1:L PR[91] R[100]mm/sec CNT100;
   1:  PR[91,1] = PR[90,1] + 60.565;
   1:  PR[91,2] = PR[90,2] + 18.606;
   1:L PR[91] R[100]mm/sec CNT100;
   1:  PR[91,1] = PR[90,1] + 55.885;
   1:  PR[91,2] = PR[90,2] + 16.778;
   1:L PR[91] R[100]mm/sec CNT100;
   1:  PR[91,1] = PR[90,1] + 51.681;
   1:  PR[91,2] = PR[90,2] + 14.184;
   1:L PR[91] R[100]mm/sec CNT100;
   1:  PR[91,1] = PR[90,1] + 50.297;
   1:  PR[91,2] = PR[90,2] + 13.161;
   1:L PR[91] R[100]mm/sec CNT100;
   1:  PR[91,1] = PR[90,1] + 48.417;
   1:  PR[91,2] = PR[90,2] + 11.199;
   1:L PR[91] R[100]mm/sec CNT100;
   1:  PR[91,1] = PR[90,1] + 46.303;
   1:  PR[91,2] = PR[90,2] + 8.631;
   1:L PR[91] R[100]mm/sec CNT100;
   1:  PR[91,1] = PR[90,1] + 43.815;
   1:  PR[91,2] = PR[90,2] + 3.885;
   1:L PR[91] R[100]mm/sec CNT100;
   1:  PR[91,1] = PR[90,1] + 41.685;
   1:  PR[91,2] = PR[90,2] + 8.704;
   1:L PR[91] R[100]mm/sec CNT100;
   1:  PR[91,1] = PR[90,1] + 41.318;
   1:  PR[91,2] = PR[90,2] + 9.380;
   1:L PR[91] R[100]mm/sec CNT100;
   1:  PR[91,1] = PR[90,1] + 40.909;
   1:  PR[91,2] = PR[90,2] + 9.927;
   1:L PR[91] R[100]mm/sec CNT100;
   1:  PR[91,1] = PR[90,1] + 38.040;
   1:  PR[91,2] = PR[90,2] + 13.576;
   1:L PR[91] R[100]mm/sec CNT100;
   1:  PR[91,1] = PR[90,1] + 33.895;
   1:  PR[91,2] = PR[90,2] + 16.707;
   1:L PR[91] R[100]mm/sec CNT100;
   1:  PR[91,1] = PR[90,1] + 29.079;
   1:  PR[91,2] = PR[90,2] + 18.676;
   1:L PR[91] R[100]mm/sec CNT100;
   1:  PR[91,1] = PR[90,1] + 23.909;
   1:  PR[91,2] = PR[90,2] + 19.344;
   1:L PR[91] R[100]mm/sec CNT100;
   1:  PR[91,1] = PR[90,1] + 18.731;
   1:  PR[91,2] = PR[90,2] + 18.658;
   1:L PR[91] R[100]mm/sec CNT100;
   1:  PR[91,1] = PR[90,1] + 13.896;
   1:  PR[91,2] = PR[90,2] + 16.659;
   1:L PR[91] R[100]mm/sec CNT100;
   1:  PR[91,1] = PR[90,1] + 9.735;
   1:  PR[91,2] = PR[90,2] + 13.476;
   1:L PR[91] R[100]mm/sec CNT100;
   1:  PR[91,1] = PR[90,1] + 6.536;
   1:  PR[91,2] = PR[90,2] + 9.323;
   1:L PR[91] R[100]mm/sec CNT100;
   1:  PR[91,1] = PR[90,1] + 4.500;
   1:  PR[91,2] = PR[90,2] + 4.453;
   1:L PR[91] R[100]mm/sec CNT100;
   1:  PR[91,1] = PR[90,1] + 4.494;
   1:  PR[91,2] = PR[90,2] + 4.429;
   1:L PR[91] R[100]mm/sec CNT100;
   1:  PR[91,1] = PR[90,1] + 3.813;
   1:  PR[91,2] = PR[90,2] + -0.613;
   1:L PR[91] R[100]mm/sec CNT100;
   1:  PR[91,2] = PR[90,2] + -0.630;
   1:L PR[91] R[100]mm/sec CNT100;
   1:  PR[91,1] = PR[90,1] + 4.449;
   1:  PR[91,2] = PR[90,2] + -5.418;
   1:L PR[91] R[100]mm/sec CNT100;
   1:  PR[91,1] = PR[90,1] + 4.467;
   1:  PR[91,2] = PR[90,2] + -5.695;
   1:L PR[91] R[100]mm/sec CNT100;
   1:  PR[91,1] = PR[90,1] + 4.495;
   1:  PR[91,2] = PR[90,2] + -5.897;
   1:L PR[91] R[100]mm/sec CNT100;
   1:  PR[91,1] = PR[90,1] + 6.537;
   1:  PR[91,2] = PR[90,2] + -10.785;
   1:L PR[91] R[100]mm/sec CNT100;
   1:  PR[91,1] = PR[90,1] + 9.746;
   1:  PR[91,2] = PR[90,2] + -14.946;
   1:L PR[91] R[100]mm/sec CNT100;
   1:  PR[91,1] = PR[90,1] + 13.914;
   1:  PR[91,2] = PR[90,2] + -18.128;
   1:L PR[91] R[100]mm/sec CNT100;
   1:  PR[91,1] = PR[90,1] + 18.756;
   1:  PR[91,2] = PR[90,2] + -20.123;
   1:L PR[91] R[100]mm/sec CNT100;
   1:  PR[91,1] = PR[90,1] + 23.939;
   1:  PR[91,2] = PR[90,2] + -20.803;
   1:L PR[91] R[100]mm/sec CNT100;
   1:  PR[91,1] = PR[90,1] + 29.112;
   1:  PR[91,2] = PR[90,2] + -20.126;
   1:L PR[91] R[100]mm/sec CNT100;
   1:  PR[91,1] = PR[90,1] + 33.928;
   1:  PR[91,2] = PR[90,2] + -18.147;
   1:L PR[91] R[100]mm/sec CNT100;
   1:  PR[91,1] = PR[90,1] + 38.068;
   1:  PR[91,2] = PR[90,2] + -15.007;
   1:L PR[91] R[100]mm/sec CNT100;
   1:  PR[91,1] = PR[90,1] + 41.323;
   1:  PR[91,2] = PR[90,2] + -10.829;
   1:L PR[91] R[100]mm/sec CNT100;
   1:  PR[91,1] = PR[90,1] + 41.633;
   1:  PR[91,2] = PR[90,2] + -10.265;
   1:L PR[91] R[100]mm/sec CNT100;
   1:  PR[91,1] = PR[90,1] + 41.768;
   1:  PR[91,2] = PR[90,2] + -9.937;
   1:L PR[91] R[100]mm/sec CNT100;
   1:  PR[91,1] = PR[90,1] + 43.847;
   1:  PR[91,2] = PR[90,2] + -5.391;
   1:L PR[91] R[100]mm/sec CNT100;
   1:  PR[91,1] = PR[90,1] + 46.344;
   1:  PR[91,2] = PR[90,2] + -10.163;
   1:L PR[91] R[100]mm/sec CNT100;
   1:  PR[91,1] = PR[90,1] + 48.448;
   1:  PR[91,2] = PR[90,2] + -12.683;
   1:L PR[91] R[100]mm/sec CNT100TB   .50sec,CALL END_PUD;
   1:  PR[92] = PR[91];
   1:  PR[92,3] = PR[92,3] + 20;
   1:J PR[92] 10% FINE;
   1:  PR[91,1] = PR[90,1] + -9.454;
   1:  PR[91,2] = PR[90,2] + -16.672;
   1:  PR[92] = PR[91];
   1:  PR[92,3] = PR[92,3] + 20;
   1:J PR[92] 10% FINE;
   1:L PR[91] R[100]mm/sec CNT100;
   1:  CALL LASER_DRAHT_START;
   1:  PR[91,1] = PR[90,1] + -7.029;
   1:  PR[91,2] = PR[90,2] + -14.701;
   1:L PR[91] R[100]mm/sec CNT100;
   1:  PR[91,1] = PR[90,1] + -6.085;
   1:  PR[91,2] = PR[90,2] + -13.824;
   1:L PR[91] R[100]mm/sec CNT100;
   1:  PR[91,1] = PR[90,1] + -3.923;
   1:  PR[91,2] = PR[90,2] + -11.032;
   1:L PR[91] R[100]mm/sec CNT100;
   1:  PR[91,1] = PR[90,1] + -3.430;
   1:  PR[91,2] = PR[90,2] + -10.299;
   1:L PR[91] R[100]mm/sec CNT100;
   1:  PR[91,1] = PR[90,1] + -1.852;
   1:  PR[91,2] = PR[90,2] + -6.817;
   1:L PR[91] R[100]mm/sec CNT100;
   1:  PR[91,1] = PR[90,1] + -1.643;
   1:  PR[91,2] = PR[90,2] + -6.258;
   1:L PR[91] R[100]mm/sec CNT100;
   1:  PR[91,1] = PR[90,1] + -0.903;
   1:  PR[91,2] = PR[90,2] + -2.322;
   1:L PR[91] R[100]mm/sec CNT100;
   1:  PR[91,1] = PR[90,1] + -0.847;
   1:  PR[91,2] = PR[90,2] + -1.858;
   1:L PR[91] R[100]mm/sec CNT100;
   1:  PR[91,1] = PR[90,1] + -0.818;
   1:  PR[91,2] = PR[90,2] + -0.821;
   1:L PR[91] R[100]mm/sec CNT100;
   1:  PR[91,1] = PR[90,1] + -0.877;
   1:  PR[91,2] = PR[90,2] + -0.329;
   1:L PR[91] R[100]mm/sec CNT100;
   1:  PR[91,1] = PR[90,1] + -0.919;
   1:  PR[91,2] = PR[90,2] + 0.936;
   1:L PR[91] R[100]mm/sec CNT100;
   1:  PR[91,1] = PR[90,1] + -1.639;
   1:  PR[91,2] = PR[90,2] + 4.785;
   1:L PR[91] R[100]mm/sec CNT100;
   1:  PR[91,1] = PR[90,1] + -1.847;
   1:  PR[91,2] = PR[90,2] + 5.344;
   1:L PR[91] R[100]mm/sec CNT100;
   1:  PR[91,1] = PR[90,1] + -3.423;
   1:  PR[91,2] = PR[90,2] + 8.829;
   1:L PR[91] R[100]mm/sec CNT100;
   1:  PR[91,1] = PR[90,1] + -3.916;
   1:  PR[91,2] = PR[90,2] + 9.561;
   1:L PR[91] R[100]mm/sec CNT100;
   1:  PR[91,1] = PR[90,1] + -6.077;
   1:  PR[91,2] = PR[90,2] + 12.357;
   1:L PR[91] R[100]mm/sec CNT100;
   1:  PR[91,1] = PR[90,1] + -7.021;
   1:  PR[91,2] = PR[90,2] + 13.233;
   1:L PR[91] R[100]mm/sec CNT100;
   1:  PR[91,1] = PR[90,1] + -9.446;
   1:  PR[91,2] = PR[90,2] + 15.208;
   1:L PR[91] R[100]mm/sec CNT100;
   1:  PR[91,1] = PR[90,1] + -10.985;
   1:  PR[91,2] = PR[90,2] + 16.095;
   1:L PR[91] R[100]mm/sec CNT100;
   1:  PR[91,1] = PR[90,1] + -13.352;
   1:  PR[91,2] = PR[90,2] + 17.268;
   1:L PR[91] R[100]mm/sec CNT100;
   1:  PR[91,1] = PR[90,1] + -15.549;
   1:  PR[91,2] = PR[90,2] + 17.949;
   1:L PR[91] R[100]mm/sec CNT100;
   1:  PR[91,1] = PR[90,1] + -17.606;
   1:  PR[91,2] = PR[90,2] + 18.453;
   1:L PR[91] R[100]mm/sec CNT100;
   1:  PR[91,1] = PR[90,1] + -20.415;
   1:  PR[91,2] = PR[90,2] + 18.686;
   1:L PR[91] R[100]mm/sec CNT100;
   1:  PR[91,1] = PR[90,1] + -22.007;
   1:  PR[91,2] = PR[90,2] + 18.725;
   1:L PR[91] R[100]mm/sec CNT100;
   1:  PR[91,1] = PR[90,1] + -25.267;
   1:  PR[91,2] = PR[90,2] + 18.283;
   1:L PR[91] R[100]mm/sec CNT100;
   1:  PR[91,1] = PR[90,1] + -26.352;
   1:  PR[91,2] = PR[90,2] + 18.074;
   1:L PR[91] R[100]mm/sec CNT100;
   1:  PR[91,1] = PR[90,1] + -29.822;
   1:  PR[91,2] = PR[90,2] + 16.806;
   1:L PR[91] R[100]mm/sec CNT100;
   1:  PR[91,1] = PR[90,1] + -30.442;
   1:  PR[91,2] = PR[90,2] + 16.541;
   1:L PR[91] R[100]mm/sec CNT100;
   1:  PR[91,1] = PR[90,1] + -33.828;
   1:  PR[91,2] = PR[90,2] + 14.379;
   1:L PR[91] R[100]mm/sec CNT100;
   1:  PR[91,1] = PR[90,1] + -34.088;
   1:  PR[91,2] = PR[90,2] + 14.194;
   1:L PR[91] R[100]mm/sec CNT100;
   1:  PR[91,1] = PR[90,1] + -37.092;
   1:  PR[91,2] = PR[90,2] + 11.178;
   1:L PR[91] R[100]mm/sec CNT100;
   1:  PR[91,1] = PR[90,1] + -37.122;
   1:  PR[91,2] = PR[90,2] + 11.145;
   1:L PR[91] R[100]mm/sec CNT100;
   1:  PR[91,1] = PR[90,1] + -39.423;
   1:  PR[91,2] = PR[90,2] + 7.491;
   1:L PR[91] R[100]mm/sec CNT100;
   1:  PR[91,1] = PR[90,1] + -40.821;
   1:  PR[91,2] = PR[90,2] + 3.489;
   1:L PR[91] R[100]mm/sec CNT100;
   1:  PR[91,1] = PR[90,1] + -41.294;
   1:  PR[91,2] = PR[90,2] + -0.729;
   1:L PR[91] R[100]mm/sec CNT100;
   1:  PR[91,1] = PR[90,1] + -40.821;
   1:  PR[91,2] = PR[90,2] + -4.948;
   1:L PR[91] R[100]mm/sec CNT100;
   1:  PR[91,1] = PR[90,1] + -39.424;
   1:  PR[91,2] = PR[90,2] + -8.948;
   1:L PR[91] R[100]mm/sec CNT100;
   1:  PR[91,1] = PR[90,1] + -37.152;
   1:  PR[91,2] = PR[90,2] + -12.572;
   1:L PR[91] R[100]mm/sec CNT100;
   1:  PR[91,1] = PR[90,1] + -37.092;
   1:  PR[91,2] = PR[90,2] + -12.637;
   1:L PR[91] R[100]mm/sec CNT100;
   1:  PR[91,1] = PR[90,1] + -34.089;
   1:  PR[91,2] = PR[90,2] + -15.652;
   1:L PR[91] R[100]mm/sec CNT100;
   1:  PR[91,1] = PR[90,1] + -33.829;
   1:  PR[91,2] = PR[90,2] + -15.837;
   1:L PR[91] R[100]mm/sec CNT100;
   1:  PR[91,1] = PR[90,1] + -30.443;
   1:  PR[91,2] = PR[90,2] + -17.999;
   1:L PR[91] R[100]mm/sec CNT100;
   1:  PR[91,1] = PR[90,1] + -29.824;
   1:  PR[91,2] = PR[90,2] + -18.264;
   1:L PR[91] R[100]mm/sec CNT100;
   1:  PR[91,1] = PR[90,1] + -26.355;
   1:  PR[91,2] = PR[90,2] + -19.532;
   1:L PR[91] R[100]mm/sec CNT100;
   1:  PR[91,1] = PR[90,1] + -25.271;
   1:  PR[91,2] = PR[90,2] + -19.742;
   1:L PR[91] R[100]mm/sec CNT100;
   1:  PR[91,1] = PR[90,1] + -22.011;
   1:  PR[91,2] = PR[90,2] + -20.183;
   1:L PR[91] R[100]mm/sec CNT100;
   1:  PR[91,1] = PR[90,1] + -20.420;
   1:  PR[91,2] = PR[90,2] + -20.145;
   1:L PR[91] R[100]mm/sec CNT100;
   1:  PR[91,1] = PR[90,1] + -17.612;
   1:  PR[91,2] = PR[90,2] + -19.913;
   1:L PR[91] R[100]mm/sec CNT100;
   1:  PR[91,1] = PR[90,1] + -15.556;
   1:  PR[91,2] = PR[90,2] + -19.411;
   1:L PR[91] R[100]mm/sec CNT100;
   1:  PR[91,1] = PR[90,1] + -13.359;
   1:  PR[91,2] = PR[90,2] + -18.730;
   1:L PR[91] R[100]mm/sec CNT100;
   1:  PR[91,1] = PR[90,1] + -10.994;
   1:  PR[91,2] = PR[90,2] + -17.559;
   1:L PR[91] R[100]mm/sec CNT100;
   1:  PR[91,1] = PR[90,1] + -9.454;
   1:  PR[91,2] = PR[90,2] + -16.672;
   1:L PR[91] R[100]mm/sec CNT100TB   .50sec,CALL END_PUD;
   1:  PR[92] = PR[91];
   1:  PR[92,3] = PR[92,3] + 20;
   1:J PR[92] 10% FINE;
   1:  PR[91,1] = PR[90,1] + -88.029;
   1:  PR[91,2] = PR[90,2] + -8.350;
   1:  PR[92] = PR[91];
   1:  PR[92,3] = PR[92,3] + 20;
   1:J PR[92] 10% FINE;
   1:L PR[91] R[100]mm/sec CNT100;
   1:  CALL LASER_DRAHT_START;
   1:  PR[91,1] = PR[90,1] + -86.008;
   1:  PR[91,2] = PR[90,2] + -11.779;
   1:L PR[91] R[100]mm/sec CNT100;
   1:  PR[91,1] = PR[90,1] + -83.287;
   1:  PR[91,2] = PR[90,2] + -14.759;
   1:L PR[91] R[100]mm/sec CNT100;
   1:  PR[91,1] = PR[90,1] + -81.620;
   1:  PR[91,2] = PR[90,2] + -15.953;
   1:L PR[91] R[100]mm/sec CNT100;
   1:  PR[91,1] = PR[90,1] + -79.957;
   1:  PR[91,2] = PR[90,2] + -17.170;
   1:L PR[91] R[100]mm/sec CNT100;
   1:  PR[91,1] = PR[90,1] + -78.462;
   1:  PR[91,2] = PR[90,2] + -17.838;
   1:L PR[91] R[100]mm/sec CNT100;
   1:  PR[91,1] = PR[90,1] + -76.161;
   1:  PR[91,2] = PR[90,2] + -18.899;
   1:L PR[91] R[100]mm/sec CNT100;
   1:  PR[91,1] = PR[90,1] + -75.053;
   1:  PR[91,2] = PR[90,2] + -19.148;
   1:L PR[91] R[100]mm/sec CNT100;
   1:  PR[91,1] = PR[90,1] + -72.032;
   1:  PR[91,2] = PR[90,2] + -19.867;
   1:L PR[91] R[100]mm/sec CNT100;
   1:  PR[91,1] = PR[90,1] + -67.747;
   1:  PR[91,2] = PR[90,2] + -20.014;
   1:L PR[91] R[100]mm/sec CNT100;
   1:  PR[91,1] = PR[90,1] + -63.770;
   1:  PR[91,2] = PR[90,2] + -19.414;
   1:L PR[91] R[100]mm/sec CNT100;
   1:  PR[91,1] = PR[90,1] + -63.237;
   1:  PR[91,2] = PR[90,2] + -19.344;
   1:L PR[91] R[100]mm/sec CNT100;
   1:  PR[91,1] = PR[90,1] + -60.243;
   1:  PR[91,2] = PR[90,2] + -18.281;
   1:L PR[91] R[100]mm/sec CNT100;
   1:  PR[91,1] = PR[90,1] + -58.938;
   1:  PR[91,2] = PR[90,2] + -17.844;
   1:L PR[91] R[100]mm/sec CNT100;
   1:  PR[91,1] = PR[90,1] + -56.976;
   1:  PR[91,2] = PR[90,2] + -16.667;
   1:L PR[91] R[100]mm/sec CNT100;
   1:  PR[91,1] = PR[90,1] + -55.044;
   1:  PR[91,2] = PR[90,2] + -15.553;
   1:L PR[91] R[100]mm/sec CNT100;
   1:  PR[91,1] = PR[90,1] + -54.023;
   1:  PR[91,2] = PR[90,2] + -14.600;
   1:L PR[91] R[100]mm/sec CNT100;
   1:  PR[91,1] = PR[90,1] + -51.746;
   1:  PR[91,2] = PR[90,2] + -12.542;
   1:L PR[91] R[100]mm/sec CNT100;
   1:  PR[91,1] = PR[90,1] + -49.244;
   1:  PR[91,2] = PR[90,2] + -8.957;
   1:L PR[91] R[100]mm/sec CNT100;
   1:  PR[91,1] = PR[90,1] + -48.966;
   1:  PR[91,2] = PR[90,2] + -8.244;
   1:L PR[91] R[100]mm/sec CNT100;
   1:  PR[91,1] = PR[90,1] + -47.558;
   1:  PR[91,2] = PR[90,2] + -4.965;
   1:L PR[91] R[100]mm/sec CNT100;
   1:  PR[91,1] = PR[90,1] + -47.541;
   1:  PR[91,2] = PR[90,2] + -4.884;
   1:L PR[91] R[100]mm/sec CNT100;
   1:  PR[91,1] = PR[90,1] + -47.031;
   1:  PR[91,2] = PR[90,2] + -1.258;
   1:L PR[91] R[100]mm/sec CNT100;
   1:  PR[91,1] = PR[90,1] + -46.998;
   1:  PR[91,2] = PR[90,2] + -0.751;
   1:L PR[91] R[100]mm/sec CNT100;
   1:  PR[91,1] = PR[90,1] + -47.139;
   1:  PR[91,2] = PR[90,2] + 0.899;
   1:L PR[91] R[100]mm/sec CNT100;
   1:  PR[91,1] = PR[90,1] + -47.483;
   1:  PR[91,2] = PR[90,2] + 3.478;
   1:L PR[91] R[100]mm/sec CNT100;
   1:  PR[91,1] = PR[90,1] + -49.116;
   1:  PR[91,2] = PR[90,2] + 7.473;
   1:L PR[91] R[100]mm/sec CNT100;
   1:  PR[91,1] = PR[90,1] + -51.731;
   1:  PR[91,2] = PR[90,2] + 11.054;
   1:L PR[91] R[100]mm/sec CNT100;
   1:  PR[91,1] = PR[90,1] + -55.180;
   1:  PR[91,2] = PR[90,2] + 14.071;
   1:L PR[91] R[100]mm/sec CNT100;
   1:  PR[91,1] = PR[90,1] + -59.022;
   1:  PR[91,2] = PR[90,2] + 16.394;
   1:L PR[91] R[100]mm/sec CNT100;
   1:  PR[91,1] = PR[90,1] + -60.143;
   1:  PR[91,2] = PR[90,2] + 16.805;
   1:L PR[91] R[100]mm/sec CNT100;
   1:  PR[91,1] = PR[90,1] + -63.226;
   1:  PR[91,2] = PR[90,2] + 17.901;
   1:L PR[91] R[100]mm/sec CNT100;
   1:  PR[91,1] = PR[90,1] + -65.755;
   1:  PR[91,2] = PR[90,2] + 18.297;
   1:L PR[91] R[100]mm/sec CNT100;
   1:  PR[91,1] = PR[90,1] + -67.635;
   1:  PR[91,2] = PR[90,2] + 18.572;
   1:L PR[91] R[100]mm/sec CNT100;
   1:  PR[91,1] = PR[90,1] + -72.070;
   1:  PR[91,2] = PR[90,2] + 18.401;
   1:L PR[91] R[100]mm/sec CNT100;
   1:  PR[91,1] = PR[90,1] + -76.284;
   1:  PR[91,2] = PR[90,2] + 17.421;
   1:L PR[91] R[100]mm/sec CNT100;
   1:  PR[91,1] = PR[90,1] + -80.042;
   1:  PR[91,2] = PR[90,2] + 15.703;
   1:L PR[91] R[100]mm/sec CNT100;
   1:  PR[91,1] = PR[90,1] + -83.337;
   1:  PR[91,2] = PR[90,2] + 13.301;
   1:L PR[91] R[100]mm/sec CNT100;
   1:  PR[91,1] = PR[90,1] + -86.038;
   1:  PR[91,2] = PR[90,2] + 10.323;
   1:L PR[91] R[100]mm/sec CNT100;
   1:  PR[91,1] = PR[90,1] + -88.043;
   1:  PR[91,2] = PR[90,2] + 6.896;
   1:L PR[91] R[100]mm/sec CNT100;
   1:  PR[91,1] = PR[90,1] + -89.276;
   1:  PR[91,2] = PR[90,2] + 3.160;
   1:L PR[91] R[100]mm/sec CNT100;
   1:  PR[91,1] = PR[90,1] + -89.474;
   1:  PR[91,2] = PR[90,2] + 1.331;
   1:L PR[91] R[100]mm/sec CNT100;
   1:  PR[91,1] = PR[90,1] + -89.593;
   1:  PR[91,2] = PR[90,2] + 0.737;
   1:L PR[91] R[100]mm/sec CNT100;
   1:  PR[91,1] = PR[90,1] + -89.750;
   1:  PR[91,2] = PR[90,2] + -0.728;
   1:L PR[91] R[100]mm/sec CNT100;
   1:  PR[91,1] = PR[90,1] + -89.512;
   1:  PR[91,2] = PR[90,2] + -2.923;
   1:L PR[91] R[100]mm/sec CNT100;
   1:  PR[91,1] = PR[90,1] + -89.395;
   1:  PR[91,2] = PR[90,2] + -3.444;
   1:L PR[91] R[100]mm/sec CNT100;
   1:  PR[91,1] = PR[90,1] + -89.270;
   1:  PR[91,2] = PR[90,2] + -4.618;
   1:L PR[91] R[100]mm/sec CNT100;
   1:  PR[91,1] = PR[90,1] + -88.029;
   1:  PR[91,2] = PR[90,2] + -8.350;
   1:L PR[91] R[100]mm/sec CNT100TB   .50sec,CALL END_PUD;
   1:  PR[92] = PR[91];
   1:  PR[92,3] = PR[92,3] + 20;
   1:J PR[92] 10% FINE;
   1:  PR[91] = PR[90];
   1:  PR[91,1] = PR[90,1] + -0.522;
   1:  PR[91,2] = PR[90,2] + -2.915;
   1:  PR[91,3] = PR[90,3] + 37.895;
   1:  PR[92] = PR[91];
   1:  PR[92,3] = PR[92,3] + 20;
   1:J PR[92] 10% FINE;
   1:L PR[91] R[100]mm/sec CNT100;
   1:  CALL LASER_DRAHT_START;
   1:  PR[91,1] = PR[90,1] + -0.041;
   1:  PR[91,2] = PR[90,2] + -0.738;
   1:L PR[91] R[100]mm/sec CNT100;
   1:  PR[91,1] = PR[90,1] + -0.527;
   1:  PR[91,2] = PR[90,2] + 1.474;
   1:L PR[91] R[100]mm/sec CNT100;
   1:  PR[91,1] = PR[90,1] + -1.184;
   1:  PR[91,2] = PR[90,2] + 4.985;
   1:L PR[91] R[100]mm/sec CNT100;
   1:  PR[91,1] = PR[90,1] + -3.026;
   1:  PR[91,2] = PR[90,2] + 9.059;
   1:L PR[91] R[100]mm/sec CNT100;
   1:  PR[91,1] = PR[90,1] + -3.149;
   1:  PR[91,2] = PR[90,2] + 9.243;
   1:L PR[91] R[100]mm/sec CNT100;
   1:  PR[91,1] = PR[90,1] + -5.733;
   1:  PR[91,2] = PR[90,2] + 12.584;
   1:L PR[91] R[100]mm/sec CNT100;
   1:  PR[91,1] = PR[90,1] + -6.200;
   1:  PR[91,2] = PR[90,2] + 13.018;
   1:L PR[91] R[100]mm/sec CNT100;
   1:  PR[91,1] = PR[90,1] + -9.149;
   1:  PR[91,2] = PR[90,2] + 15.420;
   1:L PR[91] R[100]mm/sec CNT100;
   1:  PR[91,1] = PR[90,1] + -10.140;
   1:  PR[91,2] = PR[90,2] + 15.991;
   1:L PR[91] R[100]mm/sec CNT100;
   1:  PR[91,1] = PR[90,1] + -13.096;
   1:  PR[91,2] = PR[90,2] + 17.456;
   1:L PR[91] R[100]mm/sec CNT100;
   1:  PR[91,1] = PR[90,1] + -14.710;
   1:  PR[91,2] = PR[90,2] + 17.956;
   1:L PR[91] R[100]mm/sec CNT100;
   1:  PR[91,1] = PR[90,1] + -17.382;
   1:  PR[91,2] = PR[90,2] + 18.611;
   1:L PR[91] R[100]mm/sec CNT100;
   1:  PR[91,1] = PR[90,1] + -19.608;
   1:  PR[91,2] = PR[90,2] + 18.795;
   1:L PR[91] R[100]mm/sec CNT100;
   1:  PR[91,1] = PR[90,1] + -21.806;
   1:  PR[91,2] = PR[90,2] + 18.850;
   1:L PR[91] R[100]mm/sec CNT100;
   1:  PR[91,1] = PR[90,1] + -24.514;
   1:  PR[91,2] = PR[90,2] + 18.483;
   1:L PR[91] R[100]mm/sec CNT100;
   1:  PR[91,1] = PR[90,1] + -26.166;
   1:  PR[91,2] = PR[90,2] + 18.165;
   1:L PR[91] R[100]mm/sec CNT100;
   1:  PR[91,1] = PR[90,1] + -29.138;
   1:  PR[91,2] = PR[90,2] + 17.078;
   1:L PR[91] R[100]mm/sec CNT100;
   1:  PR[91,1] = PR[90,1] + -30.262;
   1:  PR[91,2] = PR[90,2] + 16.597;
   1:L PR[91] R[100]mm/sec CNT100;
   1:  PR[91,1] = PR[90,1] + -33.224;
   1:  PR[91,2] = PR[90,2] + 14.707;
   1:L PR[91] R[100]mm/sec CNT100;
   1:  PR[91,1] = PR[90,1] + -33.909;
   1:  PR[91,2] = PR[90,2] + 14.219;
   1:L PR[91] R[100]mm/sec CNT100;
   1:  PR[91,1] = PR[90,1] + -36.573;
   1:  PR[91,2] = PR[90,2] + 11.545;
   1:L PR[91] R[100]mm/sec CNT100;
   1:  PR[91,1] = PR[90,1] + -36.939;
   1:  PR[91,2] = PR[90,2] + 11.140;
   1:L PR[91] R[100]mm/sec CNT100;
   1:  PR[91,1] = PR[90,1] + -39.097;
   1:  PR[91,2] = PR[90,2] + 7.714;
   1:L PR[91] R[100]mm/sec CNT100;
   1:  PR[91,1] = PR[90,1] + -39.232;
   1:  PR[91,2] = PR[90,2] + 7.522;
   1:L PR[91] R[100]mm/sec CNT100;
   1:  PR[91,1] = PR[90,1] + -39.236;
   1:  PR[91,2] = PR[90,2] + 7.515;
   1:L PR[91] R[100]mm/sec CNT100;
   1:  PR[91,1] = PR[90,1] + -40.509;
   1:  PR[91,2] = PR[90,2] + 3.881;
   1:L PR[91] R[100]mm/sec CNT100;
   1:  PR[91,1] = PR[90,1] + -40.607;
   1:  PR[91,2] = PR[90,2] + 3.649;
   1:L PR[91] R[100]mm/sec CNT100;
   1:  PR[91,1] = PR[90,1] + -40.744;
   1:  PR[91,2] = PR[90,2] + 3.022;
   1:L PR[91] R[100]mm/sec CNT100;
   1:  PR[91,1] = PR[90,1] + -41.056;
   1:  PR[91,2] = PR[90,2] + 0.233;
   1:L PR[91] R[100]mm/sec CNT100;
   1:  PR[91,1] = PR[90,1] + -41.129;
   1:  PR[91,2] = PR[90,2] + -0.694;
   1:L PR[91] R[100]mm/sec CNT100;
   1:  PR[91,1] = PR[90,1] + -40.889;
   1:  PR[91,2] = PR[90,2] + -2.814;
   1:L PR[91] R[100]mm/sec CNT100;
   1:  PR[91,1] = PR[90,1] + -40.727;
   1:  PR[91,2] = PR[90,2] + -4.576;
   1:L PR[91] R[100]mm/sec CNT100;
   1:  PR[91,1] = PR[90,1] + -40.583;
   1:  PR[91,2] = PR[90,2] + -5.205;
   1:L PR[91] R[100]mm/sec CNT100;
   1:  PR[91,1] = PR[90,1] + -39.505;
   1:  PR[91,2] = PR[90,2] + -8.297;
   1:L PR[91] R[100]mm/sec CNT100;
   1:  PR[91,1] = PR[90,1] + -39.270;
   1:  PR[91,2] = PR[90,2] + -8.900;
   1:L PR[91] R[100]mm/sec CNT100;
   1:  PR[91,1] = PR[90,1] + -39.153;
   1:  PR[91,2] = PR[90,2] + -9.117;
   1:L PR[91] R[100]mm/sec CNT100;
   1:  PR[91,1] = PR[90,1] + -37.113;
   1:  PR[91,2] = PR[90,2] + -12.364;
   1:L PR[91] R[100]mm/sec CNT100;
   1:  PR[91,1] = PR[90,1] + -36.976;
   1:  PR[91,2] = PR[90,2] + -12.557;
   1:L PR[91] R[100]mm/sec CNT100;
   1:  PR[91,1] = PR[90,1] + -36.574;
   1:  PR[91,2] = PR[90,2] + -13.002;
   1:L PR[91] R[100]mm/sec CNT100;
   1:  PR[91,1] = PR[90,1] + -33.910;
   1:  PR[91,2] = PR[90,2] + -15.676;
   1:L PR[91] R[100]mm/sec CNT100;
   1:  PR[91,1] = PR[90,1] + -33.226;
   1:  PR[91,2] = PR[90,2] + -16.164;
   1:L PR[91] R[100]mm/sec CNT100;
   1:  PR[91,1] = PR[90,1] + -30.265;
   1:  PR[91,2] = PR[90,2] + -18.055;
   1:L PR[91] R[100]mm/sec CNT100;
   1:  PR[91,1] = PR[90,1] + -29.142;
   1:  PR[91,2] = PR[90,2] + -18.535;
   1:L PR[91] R[100]mm/sec CNT100;
   1:  PR[91,1] = PR[90,1] + -26.170;
   1:  PR[91,2] = PR[90,2] + -19.622;
   1:L PR[91] R[100]mm/sec CNT100;
   1:  PR[91,1] = PR[90,1] + -24.520;
   1:  PR[91,2] = PR[90,2] + -19.941;
   1:L PR[91] R[100]mm/sec CNT100;
   1:  PR[91,1] = PR[90,1] + -21.812;
   1:  PR[91,2] = PR[90,2] + -20.308;
   1:L PR[91] R[100]mm/sec CNT100;
   1:  PR[91,1] = PR[90,1] + -19.616;
   1:  PR[91,2] = PR[90,2] + -20.255;
   1:L PR[91] R[100]mm/sec CNT100;
   1:  PR[91,1] = PR[90,1] + -17.389;
   1:  PR[91,2] = PR[90,2] + -20.071;
   1:L PR[91] R[100]mm/sec CNT100;
   1:  PR[91,1] = PR[90,1] + -14.720;
   1:  PR[91,2] = PR[90,2] + -19.419;
   1:L PR[91] R[100]mm/sec CNT100;
   1:  PR[91,1] = PR[90,1] + -13.105;
   1:  PR[91,2] = PR[90,2] + -18.918;
   1:L PR[91] R[100]mm/sec CNT100;
   1:  PR[91,1] = PR[90,1] + -10.151;
   1:  PR[91,2] = PR[90,2] + -17.456;
   1:L PR[91] R[100]mm/sec CNT100;
   1:  PR[91,1] = PR[90,1] + -9.159;
   1:  PR[91,2] = PR[90,2] + -16.885;
   1:L PR[91] R[100]mm/sec CNT100;
   1:  PR[91,1] = PR[90,1] + -6.210;
   1:  PR[91,2] = PR[90,2] + -14.487;
   1:L PR[91] R[100]mm/sec CNT100;
   1:  PR[91,1] = PR[90,1] + -5.742;
   1:  PR[91,2] = PR[90,2] + -14.052;
   1:L PR[91] R[100]mm/sec CNT100;
   1:  PR[91,1] = PR[90,1] + -3.158;
   1:  PR[91,2] = PR[90,2] + -10.716;
   1:L PR[91] R[100]mm/sec CNT100;
   1:  PR[91,1] = PR[90,1] + -3.034;
   1:  PR[91,2] = PR[90,2] + -10.531;
   1:L PR[91] R[100]mm/sec CNT100;
   1:  PR[91,1] = PR[90,1] + -1.189;
   1:  PR[91,2] = PR[90,2] + -6.460;
   1:L PR[91] R[100]mm/sec CNT100;
   1:  PR[91,1] = PR[90,1] + -0.522;
   1:  PR[91,2] = PR[90,2] + -2.915;
   1:L PR[91] R[100]mm/sec CNT100TB   .50sec,CALL END_PUD;
   1:  PR[92] = PR[91];
   1:  PR[92,3] = PR[92,3] + 20;
   1:J PR[92] 10% FINE;
   1:  PR[91,1] = PR[90,1] + 3.385;
   1:  PR[91,2] = PR[90,2] + -0.662;
   1:  PR[92] = PR[91];
   1:  PR[92,3] = PR[92,3] + 20;
   1:J PR[92] 10% FINE;
   1:L PR[91] R[100]mm/sec CNT100;
   1:  CALL LASER_DRAHT_START;
   1:  PR[91,1] = PR[90,1] + 3.937;
   1:  PR[91,2] = PR[90,2] + -4.586;
   1:L PR[91] R[100]mm/sec CNT100;
   1:  PR[91,1] = PR[90,1] + 4.284;
   1:  PR[91,2] = PR[90,2] + -6.155;
   1:L PR[91] R[100]mm/sec CNT100;
   1:  PR[91,1] = PR[90,1] + 5.697;
   1:  PR[91,2] = PR[90,2] + -9.537;
   1:L PR[91] R[100]mm/sec CNT100;
   1:  PR[91,1] = PR[90,1] + 6.139;
   1:  PR[91,2] = PR[90,2] + -10.641;
   1:L PR[91] R[100]mm/sec CNT100;
   1:  PR[91,1] = PR[90,1] + 6.266;
   1:  PR[91,2] = PR[90,2] + -10.893;
   1:L PR[91] R[100]mm/sec CNT100;
   1:  PR[91,1] = PR[90,1] + 9.333;
   1:  PR[91,2] = PR[90,2] + -14.856;
   1:L PR[91] R[100]mm/sec CNT100;
   1:  PR[91,1] = PR[90,1] + 9.433;
   1:  PR[91,2] = PR[90,2] + -14.999;
   1:L PR[91] R[100]mm/sec CNT100;
   1:  PR[91,1] = PR[90,1] + 9.569;
   1:  PR[91,2] = PR[90,2] + -15.142;
   1:L PR[91] R[100]mm/sec CNT100;
   1:  PR[91,1] = PR[90,1] + 13.652;
   1:  PR[91,2] = PR[90,2] + -18.238;
   1:L PR[91] R[100]mm/sec CNT100;
   1:  PR[91,1] = PR[90,1] + 13.755;
   1:  PR[91,2] = PR[90,2] + -18.302;
   1:L PR[91] R[100]mm/sec CNT100;
   1:  PR[91,1] = PR[90,1] + 18.614;
   1:  PR[91,2] = PR[90,2] + -20.286;
   1:L PR[91] R[100]mm/sec CNT100;
   1:  PR[91,1] = PR[90,1] + 23.877;
   1:  PR[91,2] = PR[90,2] + -20.954;
   1:L PR[91] R[100]mm/sec CNT100;
   1:  PR[91,1] = PR[90,1] + 29.070;
   1:  PR[91,2] = PR[90,2] + -20.267;
   1:L PR[91] R[100]mm/sec CNT100;
   1:  PR[91,1] = PR[90,1] + 33.921;
   1:  PR[91,2] = PR[90,2] + -18.278;
   1:L PR[91] R[100]mm/sec CNT100;
   1:  PR[91,1] = PR[90,1] + 38.090;
   1:  PR[91,2] = PR[90,2] + -15.120;
   1:L PR[91] R[100]mm/sec CNT100;
   1:  PR[91,1] = PR[90,1] + 41.369;
   1:  PR[91,2] = PR[90,2] + -10.919;
   1:L PR[91] R[100]mm/sec CNT100;
   1:  PR[91,1] = PR[90,1] + 42.983;
   1:  PR[91,2] = PR[90,2] + -7.976;
   1:L PR[91] R[100]mm/sec CNT100;
   1:  PR[91,1] = PR[90,1] + 45.288;
   1:  PR[91,2] = PR[90,2] + -10.358;
   1:L PR[91] R[100]mm/sec CNT100;
   1:  PR[91,1] = PR[90,1] + 47.970;
   1:  PR[91,2] = PR[90,2] + -13.572;
   1:L PR[91] R[100]mm/sec CNT100;
   1:  PR[91,1] = PR[90,1] + 48.885;
   1:  PR[91,2] = PR[90,2] + -14.529;
   1:L PR[91] R[100]mm/sec CNT100;
   1:  PR[91,1] = PR[90,1] + 51.335;
   1:  PR[91,2] = PR[90,2] + -16.321;
   1:L PR[91] R[100]mm/sec CNT100;
   1:  PR[91,1] = PR[90,1] + 54.397;
   1:  PR[91,2] = PR[90,2] + -18.210;
   1:L PR[91] R[100]mm/sec CNT100;
   1:  PR[91,1] = PR[90,1] + 55.333;
   1:  PR[91,2] = PR[90,2] + -18.619;
   1:L PR[91] R[100]mm/sec CNT100;
   1:  PR[91,1] = PR[90,1] + 57.990;
   1:  PR[91,2] = PR[90,2] + -19.512;
   1:L PR[91] R[100]mm/sec CNT100;
   1:  PR[91,1] = PR[90,1] + 60.242;
   1:  PR[91,2] = PR[90,2] + -20.391;
   1:L PR[91] R[100]mm/sec CNT100;
   1:  PR[91,1] = PR[90,1] + 60.870;
   1:  PR[91,2] = PR[90,2] + -20.545;
   1:L PR[91] R[100]mm/sec CNT100;
   1:  PR[91,1] = PR[90,1] + 65.019;
   1:  PR[91,2] = PR[90,2] + -21.162;
   1:L PR[91] R[100]mm/sec CNT100;
   1:  PR[91,1] = PR[90,1] + 67.358;
   1:  PR[91,2] = PR[90,2] + -21.246;
   1:L PR[91] R[100]mm/sec CNT100;
   1:  PR[91,1] = PR[90,1] + 69.662;
   1:  PR[91,2] = PR[90,2] + -21.085;
   1:L PR[91] R[100]mm/sec CNT100;
   1:  PR[91,1] = PR[90,1] + 73.257;
   1:  PR[91,2] = PR[90,2] + -20.487;
   1:L PR[91] R[100]mm/sec CNT100;
   1:  PR[91,1] = PR[90,1] + 74.066;
   1:  PR[91,2] = PR[90,2] + -20.249;
   1:L PR[91] R[100]mm/sec CNT100;
   1:  PR[91,1] = PR[90,1] + 78.258;
   1:  PR[91,2] = PR[90,2] + -18.646;
   1:L PR[91] R[100]mm/sec CNT100;
   1:  PR[91,1] = PR[90,1] + 82.107;
   1:  PR[91,2] = PR[90,2] + -16.130;
   1:L PR[91] R[100]mm/sec CNT100;
   1:  PR[91,1] = PR[90,1] + 85.274;
   1:  PR[91,2] = PR[90,2] + -12.918;
   1:L PR[91] R[100]mm/sec CNT100;
   1:  PR[91,1] = PR[90,1] + 87.630;
   1:  PR[91,2] = PR[90,2] + -9.162;
   1:L PR[91] R[100]mm/sec CNT100;
   1:  PR[91,1] = PR[90,1] + 88.097;
   1:  PR[91,2] = PR[90,2] + -7.845;
   1:L PR[91] R[100]mm/sec CNT100;
   1:  PR[91,1] = PR[90,1] + 89.077;
   1:  PR[91,2] = PR[90,2] + -5.041;
   1:L PR[91] R[100]mm/sec CNT100;
   1:  PR[91,1] = PR[90,1] + 89.568;
   1:  PR[91,2] = PR[90,2] + -0.729;
   1:L PR[91] R[100]mm/sec CNT100;
   1:  PR[91,1] = PR[90,1] + 89.077;
   1:  PR[91,2] = PR[90,2] + 3.581;
   1:L PR[91] R[100]mm/sec CNT100;
   1:  PR[91,1] = PR[90,1] + 87.628;
   1:  PR[91,2] = PR[90,2] + 7.706;
   1:L PR[91] R[100]mm/sec CNT100;
   1:  PR[91,1] = PR[90,1] + 85.279;
   1:  PR[91,2] = PR[90,2] + 11.451;
   1:L PR[91] R[100]mm/sec CNT100;
   1:  PR[91,1] = PR[90,1] + 84.620;
   1:  PR[91,2] = PR[90,2] + 12.107;
   1:L PR[91] R[100]mm/sec CNT100;
   1:  PR[91,1] = PR[90,1] + 82.105;
   1:  PR[91,2] = PR[90,2] + 14.672;
   1:L PR[91] R[100]mm/sec CNT100;
   1:  PR[91,1] = PR[90,1] + 78.258;
   1:  PR[91,2] = PR[90,2] + 17.187;
   1:L PR[91] R[100]mm/sec CNT100;
   1:  PR[91,1] = PR[90,1] + 74.066;
   1:  PR[91,2] = PR[90,2] + 18.790;
   1:L PR[91] R[100]mm/sec CNT100;
   1:  PR[91,1] = PR[90,1] + 73.257;
   1:  PR[91,2] = PR[90,2] + 19.028;
   1:L PR[91] R[100]mm/sec CNT100;
   1:  PR[91,1] = PR[90,1] + 69.663;
   1:  PR[91,2] = PR[90,2] + 19.626;
   1:L PR[91] R[100]mm/sec CNT100;
   1:  PR[91,1] = PR[90,1] + 67.359;
   1:  PR[91,2] = PR[90,2] + 19.787;
   1:L PR[91] R[100]mm/sec CNT100;
   1:  PR[91,1] = PR[90,1] + 65.019;
   1:  PR[91,2] = PR[90,2] + 19.703;
   1:L PR[91] R[100]mm/sec CNT100;
   1:  PR[91,1] = PR[90,1] + 60.872;
   1:  PR[91,2] = PR[90,2] + 19.086;
   1:L PR[91] R[100]mm/sec CNT100;
   1:  PR[91,1] = PR[90,1] + 60.243;
   1:  PR[91,2] = PR[90,2] + 18.933;
   1:L PR[91] R[100]mm/sec CNT100;
   1:  PR[91,1] = PR[90,1] + 57.989;
   1:  PR[91,2] = PR[90,2] + 18.053;
   1:L PR[91] R[100]mm/sec CNT100;
   1:  PR[91,1] = PR[90,1] + 55.325;
   1:  PR[91,2] = PR[90,2] + 17.158;
   1:L PR[91] R[100]mm/sec CNT100;
   1:  PR[91,1] = PR[90,1] + 54.374;
   1:  PR[91,2] = PR[90,2] + 16.739;
   1:L PR[91] R[100]mm/sec CNT100;
   1:  PR[91,1] = PR[90,1] + 51.306;
   1:  PR[91,2] = PR[90,2] + 14.848;
   1:L PR[91] R[100]mm/sec CNT100;
   1:  PR[91,1] = PR[90,1] + 48.827;
   1:  PR[91,2] = PR[90,2] + 13.016;
   1:L PR[91] R[100]mm/sec CNT100;
   1:  PR[91,1] = PR[90,1] + 47.925;
   1:  PR[91,2] = PR[90,2] + 12.075;
   1:L PR[91] R[100]mm/sec CNT100;
   1:  PR[91,1] = PR[90,1] + 45.441;
   1:  PR[91,2] = PR[90,2] + 9.058;
   1:L PR[91] R[100]mm/sec CNT100;
   1:  PR[91,1] = PR[90,1] + 42.979;
   1:  PR[91,2] = PR[90,2] + 6.500;
   1:L PR[91] R[100]mm/sec CNT100;
   1:  PR[91,1] = PR[90,1] + 41.357;
   1:  PR[91,2] = PR[90,2] + 9.483;
   1:L PR[91] R[100]mm/sec CNT100;
   1:  PR[91,1] = PR[90,1] + 41.222;
   1:  PR[91,2] = PR[90,2] + 9.669;
   1:L PR[91] R[100]mm/sec CNT100;
   1:  PR[91,1] = PR[90,1] + 38.058;
   1:  PR[91,2] = PR[90,2] + 13.693;
   1:L PR[91] R[100]mm/sec CNT100;
   1:  PR[91,1] = PR[90,1] + 33.885;
   1:  PR[91,2] = PR[90,2] + 16.840;
   1:L PR[91] R[100]mm/sec CNT100;
   1:  PR[91,1] = PR[90,1] + 29.034;
   1:  PR[91,2] = PR[90,2] + 18.817;
   1:L PR[91] R[100]mm/sec CNT100;
   1:  PR[91,1] = PR[90,1] + 23.845;
   1:  PR[91,2] = PR[90,2] + 19.495;
   1:L PR[91] R[100]mm/sec CNT100;
   1:  PR[91,1] = PR[90,1] + 18.587;
   1:  PR[91,2] = PR[90,2] + 18.820;
   1:L PR[91] R[100]mm/sec CNT100;
   1:  PR[91,1] = PR[90,1] + 13.737;
   1:  PR[91,2] = PR[90,2] + 16.833;
   1:L PR[91] R[100]mm/sec CNT100;
   1:  PR[91,1] = PR[90,1] + 13.634;
   1:  PR[91,2] = PR[90,2] + 16.769;
   1:L PR[91] R[100]mm/sec CNT100;
   1:  PR[91,1] = PR[90,1] + 9.558;
   1:  PR[91,2] = PR[90,2] + 13.673;
   1:L PR[91] R[100]mm/sec CNT100;
   1:  PR[91,1] = PR[90,1] + 9.386;
   1:  PR[91,2] = PR[90,2] + 13.492;
   1:L PR[91] R[100]mm/sec CNT100;
   1:  PR[91,1] = PR[90,1] + 6.330;
   1:  PR[91,2] = PR[90,2] + 9.542;
   1:L PR[91] R[100]mm/sec CNT100;
   1:  PR[91,1] = PR[90,1] + 6.175;
   1:  PR[91,2] = PR[90,2] + 9.261;
   1:L PR[91] R[100]mm/sec CNT100;
   1:  PR[91,1] = PR[90,1] + 4.295;
   1:  PR[91,2] = PR[90,2] + 4.736;
   1:L PR[91] R[100]mm/sec CNT100;
   1:  PR[91,1] = PR[90,1] + 3.947;
   1:  PR[91,2] = PR[90,2] + 3.180;
   1:L PR[91] R[100]mm/sec CNT100;
   1:  PR[91,1] = PR[90,1] + 3.727;
   1:  PR[91,2] = PR[90,2] + 1.543;
   1:L PR[91] R[100]mm/sec CNT100;
   1:  PR[91,1] = PR[90,1] + 3.385;
   1:  PR[91,2] = PR[90,2] + -0.662;
   1:L PR[91] R[100]mm/sec CNT100TB   .50sec,CALL END_PUD;
   1:  PR[92] = PR[91];
   1:  PR[92,3] = PR[92,3] + 20;
   1:J PR[92] 10% FINE;
   1:  PR[91,1] = PR[90,1] + -48.280;
   1:  PR[91,2] = PR[90,2] + -9.189;
   1:  PR[92] = PR[91];
   1:  PR[92,3] = PR[92,3] + 20;
   1:J PR[92] 10% FINE;
   1:L PR[91] R[100]mm/sec CNT100;
   1:  CALL LASER_DRAHT_START;
   1:  PR[91,1] = PR[90,1] + -47.842;
   1:  PR[91,2] = PR[90,2] + -8.344;
   1:L PR[91] R[100]mm/sec CNT100;
   1:  PR[91,1] = PR[90,1] + -46.537;
   1:  PR[91,2] = PR[90,2] + -5.304;
   1:L PR[91] R[100]mm/sec CNT100;
   1:  PR[91,1] = PR[90,1] + -46.350;
   1:  PR[91,2] = PR[90,2] + -4.422;
   1:L PR[91] R[100]mm/sec CNT100;
   1:  PR[91,1] = PR[90,1] + -46.052;
   1:  PR[91,2] = PR[90,2] + -2.307;
   1:L PR[91] R[100]mm/sec CNT100;
   1:  PR[91,1] = PR[90,1] + -45.952;
   1:  PR[91,2] = PR[90,2] + -0.751;
   1:L PR[91] R[100]mm/sec CNT100;
   1:  PR[91,1] = PR[90,1] + -45.988;
   1:  PR[91,2] = PR[90,2] + -0.330;
   1:L PR[91] R[100]mm/sec CNT100;
   1:  PR[91,1] = PR[90,1] + -46.502;
   1:  PR[91,2] = PR[90,2] + 3.527;
   1:L PR[91] R[100]mm/sec CNT100;
   1:  PR[91,1] = PR[90,1] + -48.161;
   1:  PR[91,2] = PR[90,2] + 7.565;
   1:L PR[91] R[100]mm/sec CNT100;
   1:  PR[91,1] = PR[90,1] + -50.814;
   1:  PR[91,2] = PR[90,2] + 11.180;
   1:L PR[91] R[100]mm/sec CNT100;
   1:  PR[91,1] = PR[90,1] + -54.291;
   1:  PR[91,2] = PR[90,2] + 14.198;
   1:L PR[91] R[100]mm/sec CNT100;
   1:  PR[91,1] = PR[90,1] + -57.643;
   1:  PR[91,2] = PR[90,2] + 16.065;
   1:L PR[91] R[100]mm/sec CNT100;
   1:  PR[91,1] = PR[90,1] + -58.400;
   1:  PR[91,2] = PR[90,2] + 16.522;
   1:L PR[91] R[100]mm/sec CNT100;
   1:  PR[91,1] = PR[90,1] + -62.648;
   1:  PR[91,2] = PR[90,2] + 18.035;
   1:L PR[91] R[100]mm/sec CNT100;
   1:  PR[91,1] = PR[90,1] + -64.155;
   1:  PR[91,2] = PR[90,2] + 18.271;
   1:L PR[91] R[100]mm/sec CNT100;
   1:  PR[91,1] = PR[90,1] + -67.091;
   1:  PR[91,2] = PR[90,2] + 18.701;
   1:L PR[91] R[100]mm/sec CNT100;
   1:  PR[91,1] = PR[90,1] + -69.914;
   1:  PR[91,2] = PR[90,2] + 18.597;
   1:L PR[91] R[100]mm/sec CNT100;
   1:  PR[91,1] = PR[90,1] + -71.543;
   1:  PR[91,2] = PR[90,2] + 18.521;
   1:L PR[91] R[100]mm/sec CNT100;
   1:  PR[91,1] = PR[90,1] + -75.829;
   1:  PR[91,2] = PR[90,2] + 17.518;
   1:L PR[91] R[100]mm/sec CNT100;
   1:  PR[91,1] = PR[90,1] + -79.715;
   1:  PR[91,2] = PR[90,2] + 15.766;
   1:L PR[91] R[100]mm/sec CNT100;
   1:  PR[91,1] = PR[90,1] + -83.016;
   1:  PR[91,2] = PR[90,2] + 13.356;
   1:L PR[91] R[100]mm/sec CNT100;
   1:  PR[91,1] = PR[90,1] + -85.724;
   1:  PR[91,2] = PR[90,2] + 10.364;
   1:L PR[91] R[100]mm/sec CNT100;
   1:  PR[91,1] = PR[90,1] + -87.735;
   1:  PR[91,2] = PR[90,2] + 6.923;
   1:L PR[91] R[100]mm/sec CNT100;
   1:  PR[91,1] = PR[90,1] + -88.971;
   1:  PR[91,2] = PR[90,2] + 3.173;
   1:L PR[91] R[100]mm/sec CNT100;
   1:  PR[91,1] = PR[90,1] + -89.113;
   1:  PR[91,2] = PR[90,2] + 1.861;
   1:L PR[91] R[100]mm/sec CNT100;
   1:  PR[91,1] = PR[90,1] + -89.201;
   1:  PR[91,2] = PR[90,2] + 1.425;
   1:L PR[91] R[100]mm/sec CNT100;
   1:  PR[91,1] = PR[90,1] + -89.431;
   1:  PR[91,2] = PR[90,2] + -0.728;
   1:L PR[91] R[100]mm/sec CNT100;
   1:  PR[91,1] = PR[90,1] + -89.263;
   1:  PR[91,2] = PR[90,2] + -2.277;
   1:L PR[91] R[100]mm/sec CNT100;
   1:  PR[91,1] = PR[90,1] + -89.103;
   1:  PR[91,2] = PR[90,2] + -2.989;
   1:L PR[91] R[100]mm/sec CNT100;
   1:  PR[91,1] = PR[90,1] + -88.928;
   1:  PR[91,2] = PR[90,2] + -4.633;
   1:L PR[91] R[100]mm/sec CNT100;
   1:  PR[91,1] = PR[90,1] + -87.684;
   1:  PR[91,2] = PR[90,2] + -8.380;
   1:L PR[91] R[100]mm/sec CNT100;
   1:  PR[91,1] = PR[90,1] + -85.656;
   1:  PR[91,2] = PR[90,2] + -11.824;
   1:L PR[91] R[100]mm/sec CNT100;
   1:  PR[91,1] = PR[90,1] + -82.928;
   1:  PR[91,2] = PR[90,2] + -14.818;
   1:L PR[91] R[100]mm/sec CNT100;
   1:  PR[91,1] = PR[90,1] + -81.651;
   1:  PR[91,2] = PR[90,2] + -15.733;
   1:L PR[91] R[100]mm/sec CNT100;
   1:  PR[91,1] = PR[90,1] + -79.588;
   1:  PR[91,2] = PR[90,2] + -17.243;
   1:L PR[91] R[100]mm/sec CNT100;
   1:  PR[91,1] = PR[90,1] + -78.546;
   1:  PR[91,2] = PR[90,2] + -17.708;
   1:L PR[91] R[100]mm/sec CNT100;
   1:  PR[91,1] = PR[90,1] + -75.767;
